ABB RAPID module: Module_OpenholeUD.modx

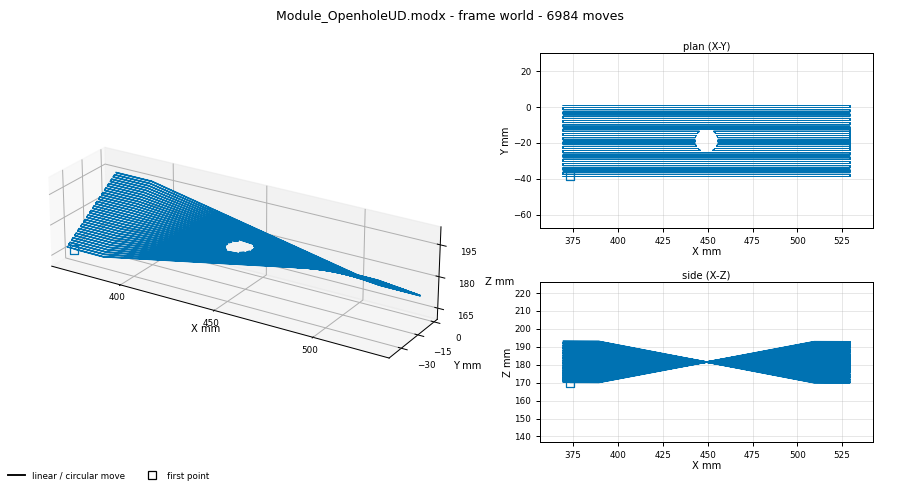
[picture p0: tool path of Module_OpenholeUD.modx in frame world, 6984 of 6984 moves have a stored position in this frame; points joined in program order, loops and branches not executed]
MODULE Module_OpenholeUD

	VAR robtarget OpenholeUD_0 := [[373.31, -38.7, 169.95], [-0.183051, 0.683002, 0.683002, 0.183051], [0,0,0,0], [9E9, 9E9, 9E9, 9E9, 9E9, 9E9]];
	VAR robtarget OpenholeUD_1 := [[377.31, -38.7, 169.94], [-0.183051, 0.683002, 0.683002, 0.183051], [0,0,0,0], [9E9, 9E9, 9E9, 9E9, 9E9, 9E9]];
	VAR robtarget OpenholeUD_2 := [[381.31, -38.7, 169.93], [-0.183051, 0.683002, 0.683002, 0.183051], [0,0,0,0], [9E9, 9E9, 9E9, 9E9, 9E9, 9E9]];
	VAR robtarget OpenholeUD_3 := [[385.31, -38.7, 169.91], [-0.183051, 0.683002, 0.683002, 0.183051], [0,0,0,0], [9E9, 9E9, 9E9, 9E9, 9E9, 9E9]];
	VAR robtarget OpenholeUD_4 := [[389.31, -38.7, 169.9], [-0.126214, 0.695751, 0.665684, 0.238465], [0,0,0,0], [9E9, 9E9, 9E9, 9E9, 9E9, 9E9]];
	VAR robtarget OpenholeUD_5 := [[393.24, -38.7, 170.64], [-0.115233, 0.697654, 0.668744, 0.229742], [0,0,0,0], [9E9, 9E9, 9E9, 9E9, 9E9, 9E9]];
	VAR robtarget OpenholeUD_6 := [[397.17, -38.7, 171.39], [-0.103921, 0.699429, 0.671799, 0.220649], [0,0,0,0], [9E9, 9E9, 9E9, 9E9, 9E9, 9E9]];
	VAR robtarget OpenholeUD_7 := [[401.1, -38.7, 172.13], [-0.092289, 0.701058, 0.674835, 0.211182], [0,0,0,0], [9E9, 9E9, 9E9, 9E9, 9E9, 9E9]];
	VAR robtarget OpenholeUD_8 := [[405.03, -38.7, 172.88], [-0.080349, 0.702527, 0.677838, 0.201336], [0,0,0,0], [9E9, 9E9, 9E9, 9E9, 9E9, 9E9]];
	VAR robtarget OpenholeUD_9 := [[408.96, -38.7, 173.62], [-0.068121, 0.703818, 0.680791, 0.191112], [0,0,0,0], [9E9, 9E9, 9E9, 9E9, 9E9, 9E9]];
	VAR robtarget OpenholeUD_10 := [[412.89, -38.7, 174.36], [-0.055624, 0.704916, 0.683677, 0.180513], [0,0,0,0], [9E9, 9E9, 9E9, 9E9, 9E9, 9E9]];
	VAR robtarget OpenholeUD_11 := [[416.82, -38.7, 175.11], [-0.042884, 0.705805, 0.68648, 0.169546], [0,0,0,0], [9E9, 9E9, 9E9, 9E9, 9E9, 9E9]];
	VAR robtarget OpenholeUD_12 := [[420.75, -38.7, 175.85], [-0.029931, 0.706473, 0.689178, 0.15822], [0,0,0,0], [9E9, 9E9, 9E9, 9E9, 9E9, 9E9]];
	VAR robtarget OpenholeUD_13 := [[424.68, -38.7, 176.59], [-0.016796, 0.706907, 0.691754, 0.14655], [0,0,0,0], [9E9, 9E9, 9E9, 9E9, 9E9, 9E9]];
	VAR robtarget OpenholeUD_14 := [[428.61, -38.7, 177.34], [-0.003517, 0.707098, 0.694187, 0.134555], [0,0,0,0], [9E9, 9E9, 9E9, 9E9, 9E9, 9E9]];
	VAR robtarget OpenholeUD_15 := [[432.54, -38.7, 178.08], [0.009868, 0.707038, 0.696458, 0.122257], [0,0,0,0], [9E9, 9E9, 9E9, 9E9, 9E9, 9E9]];
	VAR robtarget OpenholeUD_16 := [[436.47, -38.7, 178.83], [0.023319, 0.706722, 0.698548, 0.109684], [0,0,0,0], [9E9, 9E9, 9E9, 9E9, 9E9, 9E9]];
	VAR robtarget OpenholeUD_17 := [[440.4, -38.7, 179.57], [0.03679, 0.706149, 0.700441, 0.096866], [0,0,0,0], [9E9, 9E9, 9E9, 9E9, 9E9, 9E9]];
	VAR robtarget OpenholeUD_18 := [[444.33, -38.7, 180.31], [0.05024, 0.70532, 0.702119, 0.083838], [0,0,0,0], [9E9, 9E9, 9E9, 9E9, 9E9, 9E9]];
	VAR robtarget OpenholeUD_19 := [[448.26, -38.7, 181.06], [0.063624, 0.704239, 0.70357, 0.070638], [0,0,0,0], [9E9, 9E9, 9E9, 9E9, 9E9, 9E9]];
	VAR robtarget OpenholeUD_20 := [[452.19, -38.7, 181.8], [0.076899, 0.702913, 0.704781, 0.057307], [0,0,0,0], [9E9, 9E9, 9E9, 9E9, 9E9, 9E9]];
	VAR robtarget OpenholeUD_21 := [[456.12, -38.7, 182.54], [0.090023, 0.701353, 0.705744, 0.043887], [0,0,0,0], [9E9, 9E9, 9E9, 9E9, 9E9, 9E9]];
	VAR robtarget OpenholeUD_22 := [[460.05, -38.7, 183.29], [0.102957, 0.699571, 0.706452, 0.030421], [0,0,0,0], [9E9, 9E9, 9E9, 9E9, 9E9, 9E9]];
	VAR robtarget OpenholeUD_23 := [[463.98, -38.7, 184.03], [0.115664, 0.697583, 0.706903, 0.016955], [0,0,0,0], [9E9, 9E9, 9E9, 9E9, 9E9, 9E9]];
	VAR robtarget OpenholeUD_24 := [[467.91, -38.7, 184.78], [0.128112, 0.695404, 0.707098, 0.003531], [0,0,0,0], [9E9, 9E9, 9E9, 9E9, 9E9, 9E9]];
	VAR robtarget OpenholeUD_25 := [[471.85, -38.7, 185.52], [0.14027, 0.693054, 0.707039, -0.009809], [0,0,0,0], [9E9, 9E9, 9E9, 9E9, 9E9, 9E9]];
	VAR robtarget OpenholeUD_26 := [[475.78, -38.7, 186.26], [0.152115, 0.690551, 0.706732, -0.023024], [0,0,0,0], [9E9, 9E9, 9E9, 9E9, 9E9, 9E9]];
	VAR robtarget OpenholeUD_27 := [[479.71, -38.7, 187.01], [0.163624, 0.687915, 0.706186, -0.036076], [0,0,0,0], [9E9, 9E9, 9E9, 9E9, 9E9, 9E9]];
	VAR robtarget OpenholeUD_28 := [[483.64, -38.7, 187.75], [0.174782, 0.685165, 0.705412, -0.048932], [0,0,0,0], [9E9, 9E9, 9E9, 9E9, 9E9, 9E9]];
	VAR robtarget OpenholeUD_29 := [[487.57, -38.7, 188.49], [0.185577, 0.68232, 0.704422, -0.06156], [0,0,0,0], [9E9, 9E9, 9E9, 9E9, 9E9, 9E9]];
	VAR robtarget OpenholeUD_30 := [[491.5, -38.7, 189.24], [0.195999, 0.6794, 0.703231, -0.073932], [0,0,0,0], [9E9, 9E9, 9E9, 9E9, 9E9, 9E9]];
	VAR robtarget OpenholeUD_31 := [[495.43, -38.7, 189.98], [0.206044, 0.676421, 0.701854, -0.086026], [0,0,0,0], [9E9, 9E9, 9E9, 9E9, 9E9, 9E9]];
	VAR robtarget OpenholeUD_32 := [[499.36, -38.7, 190.73], [0.215711, 0.673401, 0.700308, -0.097822], [0,0,0,0], [9E9, 9E9, 9E9, 9E9, 9E9, 9E9]];
	VAR robtarget OpenholeUD_33 := [[503.29, -38.7, 191.47], [0.225001, 0.670354, 0.698608, -0.109304], [0,0,0,0], [9E9, 9E9, 9E9, 9E9, 9E9, 9E9]];
	VAR robtarget OpenholeUD_34 := [[509.38, -38.7, 192.62], [0.183051, 0.683002, 0.683002, -0.183051], [0,0,0,0], [9E9, 9E9, 9E9, 9E9, 9E9, 9E9]];
	VAR robtarget OpenholeUD_35 := [[513.38, -38.7, 192.61], [0.183051, 0.683002, 0.683002, -0.183051], [0,0,0,0], [9E9, 9E9, 9E9, 9E9, 9E9, 9E9]];
	VAR robtarget OpenholeUD_36 := [[517.38, -38.7, 192.6], [0.183051, 0.683002, 0.683002, -0.183051], [0,0,0,0], [9E9, 9E9, 9E9, 9E9, 9E9, 9E9]];
	VAR robtarget OpenholeUD_37 := [[521.38, -38.7, 192.59], [0.183051, 0.683002, 0.683002, -0.183051], [0,0,0,0], [9E9, 9E9, 9E9, 9E9, 9E9, 9E9]];
	VAR robtarget OpenholeUD_38 := [[529.38, -38.7, 192.56], [0.183051, 0.683002, 0.683002, -0.183051], [0,0,0,0], [9E9, 9E9, 9E9, 9E9, 9E9, 9E9]];
	VAR robtarget OpenholeUD_39 := [[529.38, -38.7, 192.56], [0.183051, 0.683002, 0.683002, -0.183051], [0,0,0,0], [9E9, 9E9, 9E9, 9E9, 9E9, 9E9]];
	VAR robtarget OpenholeUD_40 := [[529.38, -37.5, 191.87], [0.183051, 0.683002, 0.683002, -0.183051], [0,0,0,0], [9E9, 9E9, 9E9, 9E9, 9E9, 9E9]];
	VAR robtarget OpenholeUD_41 := [[525.38, -37.5, 191.88], [0.183051, 0.683002, 0.683002, -0.183051], [0,0,0,0], [9E9, 9E9, 9E9, 9E9, 9E9, 9E9]];
	VAR robtarget OpenholeUD_42 := [[521.38, -37.5, 191.89], [0.183051, 0.683002, 0.683002, -0.183051], [0,0,0,0], [9E9, 9E9, 9E9, 9E9, 9E9, 9E9]];
	VAR robtarget OpenholeUD_43 := [[517.38, -37.5, 191.9], [0.183051, 0.683002, 0.683002, -0.183051], [0,0,0,0], [9E9, 9E9, 9E9, 9E9, 9E9, 9E9]];
	VAR robtarget OpenholeUD_44 := [[509.38, -37.5, 191.93], [0.183051, 0.683002, 0.683002, -0.183051], [0,0,0,0], [9E9, 9E9, 9E9, 9E9, 9E9, 9E9]];
	VAR robtarget OpenholeUD_45 := [[505.44, -37.5, 191.23], [0.226628, 0.669806, 0.697036, -0.118915], [0,0,0,0], [9E9, 9E9, 9E9, 9E9, 9E9, 9E9]];
	VAR robtarget OpenholeUD_46 := [[501.5, -37.5, 190.53], [0.21746, 0.672838, 0.698865, -0.107647], [0,0,0,0], [9E9, 9E9, 9E9, 9E9, 9E9, 9E9]];
	VAR robtarget OpenholeUD_47 := [[497.56, -37.5, 189.83], [0.207916, 0.675848, 0.700552, -0.096055], [0,0,0,0], [9E9, 9E9, 9E9, 9E9, 9E9, 9E9]];
	VAR robtarget OpenholeUD_48 := [[493.63, -37.5, 189.13], [0.197995, 0.678821, 0.702082, -0.084152], [0,0,0,0], [9E9, 9E9, 9E9, 9E9, 9E9, 9E9]];
	VAR robtarget OpenholeUD_49 := [[489.69, -37.5, 188.43], [0.187696, 0.681741, 0.703436, -0.071954], [0,0,0,0], [9E9, 9E9, 9E9, 9E9, 9E9, 9E9]];
	VAR robtarget OpenholeUD_50 := [[485.75, -37.5, 187.73], [0.177023, 0.68459, 0.7046, -0.059484], [0,0,0,0], [9E9, 9E9, 9E9, 9E9, 9E9, 9E9]];
	VAR robtarget OpenholeUD_51 := [[481.81, -37.5, 187.03], [0.165982, 0.68735, 0.705559, -0.046765], [0,0,0,0], [9E9, 9E9, 9E9, 9E9, 9E9, 9E9]];
	VAR robtarget OpenholeUD_52 := [[477.87, -37.5, 186.33], [0.154586, 0.690002, 0.706297, -0.033827], [0,0,0,0], [9E9, 9E9, 9E9, 9E9, 9E9, 9E9]];
	VAR robtarget OpenholeUD_53 := [[473.94, -37.5, 185.63], [0.142847, 0.692528, 0.706804, -0.020702], [0,0,0,0], [9E9, 9E9, 9E9, 9E9, 9E9, 9E9]];
	VAR robtarget OpenholeUD_54 := [[470, -37.5, 184.93], [0.130787, 0.694906, 0.707068, -0.007426], [0,0,0,0], [9E9, 9E9, 9E9, 9E9, 9E9, 9E9]];
	VAR robtarget OpenholeUD_55 := [[466.06, -37.5, 184.23], [0.118427, 0.697119, 0.707082, 0.005963], [0,0,0,0], [9E9, 9E9, 9E9, 9E9, 9E9, 9E9]];
	VAR robtarget OpenholeUD_56 := [[462.12, -37.5, 183.53], [0.105796, 0.699147, 0.70684, 0.019422], [0,0,0,0], [9E9, 9E9, 9E9, 9E9, 9E9, 9E9]];
	VAR robtarget OpenholeUD_57 := [[458.18, -37.5, 182.83], [0.092926, 0.700974, 0.706341, 0.03291], [0,0,0,0], [9E9, 9E9, 9E9, 9E9, 9E9, 9E9]];
	VAR robtarget OpenholeUD_58 := [[454.24, -37.5, 182.13], [0.079851, 0.702584, 0.705584, 0.046383], [0,0,0,0], [9E9, 9E9, 9E9, 9E9, 9E9, 9E9]];
	VAR robtarget OpenholeUD_59 := [[450.31, -37.5, 181.43], [0.06661, 0.703962, 0.704574, 0.059795], [0,0,0,0], [9E9, 9E9, 9E9, 9E9, 9E9, 9E9]];
	VAR robtarget OpenholeUD_60 := [[446.37, -37.5, 180.73], [0.053244, 0.705099, 0.703318, 0.073104], [0,0,0,0], [9E9, 9E9, 9E9, 9E9, 9E9, 9E9]];
	VAR robtarget OpenholeUD_61 := [[442.43, -37.5, 180.03], [0.039796, 0.705986, 0.701825, 0.086268], [0,0,0,0], [9E9, 9E9, 9E9, 9E9, 9E9, 9E9]];
	VAR robtarget OpenholeUD_62 := [[438.49, -37.5, 179.33], [0.02631, 0.706617, 0.700107, 0.099247], [0,0,0,0], [9E9, 9E9, 9E9, 9E9, 9E9, 9E9]];
	VAR robtarget OpenholeUD_63 := [[434.55, -37.5, 178.63], [0.012829, 0.70699, 0.69818, 0.112004], [0,0,0,0], [9E9, 9E9, 9E9, 9E9, 9E9, 9E9]];
	VAR robtarget OpenholeUD_64 := [[430.61, -37.5, 177.93], [-0.000601, 0.707107, 0.696059, 0.124505], [0,0,0,0], [9E9, 9E9, 9E9, 9E9, 9E9, 9E9]];
	VAR robtarget OpenholeUD_65 := [[426.68, -37.5, 177.23], [-0.013941, 0.706969, 0.693763, 0.136721], [0,0,0,0], [9E9, 9E9, 9E9, 9E9, 9E9, 9E9]];
	VAR robtarget OpenholeUD_66 := [[422.74, -37.5, 176.53], [-0.027148, 0.706585, 0.691311, 0.148626], [0,0,0,0], [9E9, 9E9, 9E9, 9E9, 9E9, 9E9]];
	VAR robtarget OpenholeUD_67 := [[418.8, -37.5, 175.83], [-0.040187, 0.705964, 0.688721, 0.160199], [0,0,0,0], [9E9, 9E9, 9E9, 9E9, 9E9, 9E9]];
	VAR robtarget OpenholeUD_68 := [[414.86, -37.5, 175.13], [-0.053022, 0.705116, 0.686013, 0.171422], [0,0,0,0], [9E9, 9E9, 9E9, 9E9, 9E9, 9E9]];
	VAR robtarget OpenholeUD_69 := [[410.92, -37.5, 174.43], [-0.065623, 0.704055, 0.683208, 0.182284], [0,0,0,0], [9E9, 9E9, 9E9, 9E9, 9E9, 9E9]];
	VAR robtarget OpenholeUD_70 := [[406.98, -37.5, 173.73], [-0.077963, 0.702796, 0.680322, 0.192774], [0,0,0,0], [9E9, 9E9, 9E9, 9E9, 9E9, 9E9]];
	VAR robtarget OpenholeUD_71 := [[403.05, -37.5, 173.03], [-0.09002, 0.701353, 0.677374, 0.202889], [0,0,0,0], [9E9, 9E9, 9E9, 9E9, 9E9, 9E9]];
	VAR robtarget OpenholeUD_72 := [[399.11, -37.5, 172.33], [-0.101773, 0.699744, 0.674382, 0.212625], [0,0,0,0], [9E9, 9E9, 9E9, 9E9, 9E9, 9E9]];
	VAR robtarget OpenholeUD_73 := [[395.17, -37.5, 171.63], [-0.113209, 0.697986, 0.671359, 0.221984], [0,0,0,0], [9E9, 9E9, 9E9, 9E9, 9E9, 9E9]];
	VAR robtarget OpenholeUD_74 := [[389.31, -37.5, 170.59], [-0.129603, 0.695128, 0.666839, 0.235215], [0,0,0,0], [9E9, 9E9, 9E9, 9E9, 9E9, 9E9]];
	VAR robtarget OpenholeUD_75 := [[385.31, -37.5, 170.61], [-0.183051, 0.683002, 0.683002, 0.183051], [0,0,0,0], [9E9, 9E9, 9E9, 9E9, 9E9, 9E9]];
	VAR robtarget OpenholeUD_76 := [[381.31, -37.5, 170.62], [-0.183051, 0.683002, 0.683002, 0.183051], [0,0,0,0], [9E9, 9E9, 9E9, 9E9, 9E9, 9E9]];
	VAR robtarget OpenholeUD_77 := [[377.31, -37.5, 170.63], [-0.183051, 0.683002, 0.683002, 0.183051], [0,0,0,0], [9E9, 9E9, 9E9, 9E9, 9E9, 9E9]];
	VAR robtarget OpenholeUD_78 := [[373.31, -37.5, 170.64], [-0.183051, 0.683002, 0.683002, 0.183051], [0,0,0,0], [9E9, 9E9, 9E9, 9E9, 9E9, 9E9]];
	VAR robtarget OpenholeUD_79 := [[369.31, -37.5, 170.66], [-0.183051, 0.683002, 0.683002, 0.183051], [0,0,0,0], [9E9, 9E9, 9E9, 9E9, 9E9, 9E9]];
	VAR robtarget OpenholeUD_80 := [[369.31, -37.5, 170.66], [-0.183051, 0.683002, 0.683002, 0.183051], [0,0,0,0], [9E9, 9E9, 9E9, 9E9, 9E9, 9E9]];
	VAR robtarget OpenholeUD_81 := [[369.31, -36.3, 171.35], [-0.183051, 0.683002, 0.683002, 0.183051], [0,0,0,0], [9E9, 9E9, 9E9, 9E9, 9E9, 9E9]];
	VAR robtarget OpenholeUD_82 := [[373.31, -36.3, 171.34], [-0.183051, 0.683002, 0.683002, 0.183051], [0,0,0,0], [9E9, 9E9, 9E9, 9E9, 9E9, 9E9]];
	VAR robtarget OpenholeUD_83 := [[377.31, -36.3, 171.32], [-0.183051, 0.683002, 0.683002, 0.183051], [0,0,0,0], [9E9, 9E9, 9E9, 9E9, 9E9, 9E9]];
	VAR robtarget OpenholeUD_84 := [[381.31, -36.3, 171.31], [-0.183051, 0.683002, 0.683002, 0.183051], [0,0,0,0], [9E9, 9E9, 9E9, 9E9, 9E9, 9E9]];
	VAR robtarget OpenholeUD_85 := [[385.31, -36.3, 171.3], [-0.183051, 0.683002, 0.683002, 0.183051], [0,0,0,0], [9E9, 9E9, 9E9, 9E9, 9E9, 9E9]];
	VAR robtarget OpenholeUD_86 := [[389.31, -36.3, 171.29], [-0.133, 0.694486, 0.667982, 0.23195], [0,0,0,0], [9E9, 9E9, 9E9, 9E9, 9E9, 9E9]];
	VAR robtarget OpenholeUD_87 := [[393.26, -36.3, 171.94], [-0.122099, 0.696485, 0.671002, 0.22306], [0,0,0,0], [9E9, 9E9, 9E9, 9E9, 9E9, 9E9]];
	VAR robtarget OpenholeUD_88 := [[397.21, -36.3, 172.6], [-0.11086, 0.698362, 0.67401, 0.213799], [0,0,0,0], [9E9, 9E9, 9E9, 9E9, 9E9, 9E9]];
	VAR robtarget OpenholeUD_89 := [[401.15, -36.3, 173.25], [-0.099295, 0.7001, 0.676992, 0.204163], [0,0,0,0], [9E9, 9E9, 9E9, 9E9, 9E9, 9E9]];
	VAR robtarget OpenholeUD_90 := [[405.1, -36.3, 173.91], [-0.087415, 0.701683, 0.679931, 0.194149], [0,0,0,0], [9E9, 9E9, 9E9, 9E9, 9E9, 9E9]];
	VAR robtarget OpenholeUD_91 := [[409.04, -36.3, 174.56], [-0.075237, 0.703093, 0.682813, 0.183758], [0,0,0,0], [9E9, 9E9, 9E9, 9E9, 9E9, 9E9]];
	VAR robtarget OpenholeUD_92 := [[412.99, -36.3, 175.22], [-0.062782, 0.704314, 0.685619, 0.172994], [0,0,0,0], [9E9, 9E9, 9E9, 9E9, 9E9, 9E9]];
	VAR robtarget OpenholeUD_93 := [[416.94, -36.3, 175.88], [-0.050075, 0.705331, 0.688331, 0.161866], [0,0,0,0], [9E9, 9E9, 9E9, 9E9, 9E9, 9E9]];
	VAR robtarget OpenholeUD_94 := [[420.88, -36.3, 176.53], [-0.037144, 0.706131, 0.69093, 0.150384], [0,0,0,0], [9E9, 9E9, 9E9, 9E9, 9E9, 9E9]];
	VAR robtarget OpenholeUD_95 := [[424.83, -36.3, 177.19], [-0.024021, 0.706699, 0.693397, 0.138564], [0,0,0,0], [9E9, 9E9, 9E9, 9E9, 9E9, 9E9]];
	VAR robtarget OpenholeUD_96 := [[428.77, -36.3, 177.84], [-0.010743, 0.707025, 0.695713, 0.126426], [0,0,0,0], [9E9, 9E9, 9E9, 9E9, 9E9, 9E9]];
	VAR robtarget OpenholeUD_97 := [[432.72, -36.3, 178.5], [0.002652, 0.707102, 0.697858, 0.113995], [0,0,0,0], [9E9, 9E9, 9E9, 9E9, 9E9, 9E9]];
	VAR robtarget OpenholeUD_98 := [[436.67, -36.3, 179.15], [0.016123, 0.706923, 0.699813, 0.101298], [0,0,0,0], [9E9, 9E9, 9E9, 9E9, 9E9, 9E9]];
	VAR robtarget OpenholeUD_99 := [[440.61, -36.3, 179.81], [0.029627, 0.706486, 0.701563, 0.088368], [0,0,0,0], [9E9, 9E9, 9E9, 9E9, 9E9, 9E9]];
	VAR robtarget OpenholeUD_100 := [[444.56, -36.3, 180.47], [0.04312, 0.705791, 0.703092, 0.075241], [0,0,0,0], [9E9, 9E9, 9E9, 9E9, 9E9, 9E9]];
	VAR robtarget OpenholeUD_101 := [[448.5, -36.3, 181.12], [0.056557, 0.704841, 0.704387, 0.061957], [0,0,0,0], [9E9, 9E9, 9E9, 9E9, 9E9, 9E9]];
	VAR robtarget OpenholeUD_102 := [[452.45, -36.3, 181.78], [0.069895, 0.703644, 0.705438, 0.048555], [0,0,0,0], [9E9, 9E9, 9E9, 9E9, 9E9, 9E9]];
	VAR robtarget OpenholeUD_103 := [[456.39, -36.3, 182.43], [0.083091, 0.702208, 0.706236, 0.03508], [0,0,0,0], [9E9, 9E9, 9E9, 9E9, 9E9, 9E9]];
	VAR robtarget OpenholeUD_104 := [[460.34, -36.3, 183.09], [0.096106, 0.700545, 0.706778, 0.021577], [0,0,0,0], [9E9, 9E9, 9E9, 9E9, 9E9, 9E9]];
	VAR robtarget OpenholeUD_105 := [[464.29, -36.3, 183.74], [0.108902, 0.69867, 0.707061, 0.008088], [0,0,0,0], [9E9, 9E9, 9E9, 9E9, 9E9, 9E9]];
	VAR robtarget OpenholeUD_106 := [[468.23, -36.3, 184.4], [0.121445, 0.6966, 0.707087, -0.005342], [0,0,0,0], [9E9, 9E9, 9E9, 9E9, 9E9, 9E9]];
	VAR robtarget OpenholeUD_107 := [[472.18, -36.3, 185.06], [0.133705, 0.694351, 0.70686, -0.018672], [0,0,0,0], [9E9, 9E9, 9E9, 9E9, 9E9, 9E9]];
	VAR robtarget OpenholeUD_108 := [[476.12, -36.3, 185.71], [0.145657, 0.691942, 0.706389, -0.031861], [0,0,0,0], [9E9, 9E9, 9E9, 9E9, 9E9, 9E9]];
	VAR robtarget OpenholeUD_109 := [[480.07, -36.3, 186.37], [0.157278, 0.689394, 0.705682, -0.044873], [0,0,0,0], [9E9, 9E9, 9E9, 9E9, 9E9, 9E9]];
	VAR robtarget OpenholeUD_110 := [[484.02, -36.3, 187.02], [0.168551, 0.686724, 0.704751, -0.057673], [0,0,0,0], [9E9, 9E9, 9E9, 9E9, 9E9, 9E9]];
	VAR robtarget OpenholeUD_111 := [[487.96, -36.3, 187.68], [0.179463, 0.683954, 0.70361, -0.070232], [0,0,0,0], [9E9, 9E9, 9E9, 9E9, 9E9, 9E9]];
	VAR robtarget OpenholeUD_112 := [[491.91, -36.3, 188.33], [0.190006, 0.6811, 0.702275, -0.082524], [0,0,0,0], [9E9, 9E9, 9E9, 9E9, 9E9, 9E9]];
	VAR robtarget OpenholeUD_113 := [[495.85, -36.3, 188.99], [0.200172, 0.678182, 0.70076, -0.094526], [0,0,0,0], [9E9, 9E9, 9E9, 9E9, 9E9, 9E9]];
	VAR robtarget OpenholeUD_114 := [[499.8, -36.3, 189.65], [0.209961, 0.675216, 0.699083, -0.10622], [0,0,0,0], [9E9, 9E9, 9E9, 9E9, 9E9, 9E9]];
	VAR robtarget OpenholeUD_115 := [[503.75, -36.3, 190.3], [0.219374, 0.672217, 0.69726, -0.117592], [0,0,0,0], [9E9, 9E9, 9E9, 9E9, 9E9, 9E9]];
	VAR robtarget OpenholeUD_116 := [[509.38, -36.3, 191.24], [0.183051, 0.683002, 0.683002, -0.183051], [0,0,0,0], [9E9, 9E9, 9E9, 9E9, 9E9, 9E9]];
	VAR robtarget OpenholeUD_117 := [[513.38, -36.3, 191.22], [0.183051, 0.683002, 0.683002, -0.183051], [0,0,0,0], [9E9, 9E9, 9E9, 9E9, 9E9, 9E9]];
	VAR robtarget OpenholeUD_118 := [[517.38, -36.3, 191.21], [0.183051, 0.683002, 0.683002, -0.183051], [0,0,0,0], [9E9, 9E9, 9E9, 9E9, 9E9, 9E9]];
	VAR robtarget OpenholeUD_119 := [[521.38, -36.3, 191.2], [0.183051, 0.683002, 0.683002, -0.183051], [0,0,0,0], [9E9, 9E9, 9E9, 9E9, 9E9, 9E9]];
	VAR robtarget OpenholeUD_120 := [[525.38, -36.3, 191.19], [0.183051, 0.683002, 0.683002, -0.183051], [0,0,0,0], [9E9, 9E9, 9E9, 9E9, 9E9, 9E9]];
	VAR robtarget OpenholeUD_121 := [[529.38, -36.3, 191.17], [0.183051, 0.683002, 0.683002, -0.183051], [0,0,0,0], [9E9, 9E9, 9E9, 9E9, 9E9, 9E9]];
	VAR robtarget OpenholeUD_122 := [[529.38, -36.3, 191.17], [0.183051, 0.683002, 0.683002, -0.183051], [0,0,0,0], [9E9, 9E9, 9E9, 9E9, 9E9, 9E9]];
	VAR robtarget OpenholeUD_123 := [[529.38, -35.1, 190.48], [0.183051, 0.683002, 0.683002, -0.183051], [0,0,0,0], [9E9, 9E9, 9E9, 9E9, 9E9, 9E9]];
	VAR robtarget OpenholeUD_124 := [[525.38, -35.1, 190.49], [0.183051, 0.683002, 0.683002, -0.183051], [0,0,0,0], [9E9, 9E9, 9E9, 9E9, 9E9, 9E9]];
	VAR robtarget OpenholeUD_125 := [[521.38, -35.1, 190.51], [0.183051, 0.683002, 0.683002, -0.183051], [0,0,0,0], [9E9, 9E9, 9E9, 9E9, 9E9, 9E9]];
	VAR robtarget OpenholeUD_126 := [[517.38, -35.1, 190.52], [0.183051, 0.683002, 0.683002, -0.183051], [0,0,0,0], [9E9, 9E9, 9E9, 9E9, 9E9, 9E9]];
	VAR robtarget OpenholeUD_127 := [[513.38, -35.1, 190.53], [0.183051, 0.683002, 0.683002, -0.183051], [0,0,0,0], [9E9, 9E9, 9E9, 9E9, 9E9, 9E9]];
	VAR robtarget OpenholeUD_128 := [[509.38, -35.1, 190.54], [0.183051, 0.683002, 0.683002, -0.183051], [0,0,0,0], [9E9, 9E9, 9E9, 9E9, 9E9, 9E9]];
	VAR robtarget OpenholeUD_129 := [[505.42, -35.1, 189.93], [0.219922, 0.672037, 0.695827, -0.125794], [0,0,0,0], [9E9, 9E9, 9E9, 9E9, 9E9, 9E9]];
	VAR robtarget OpenholeUD_130 := [[501.47, -35.1, 189.32], [0.210587, 0.675021, 0.697758, -0.114605], [0,0,0,0], [9E9, 9E9, 9E9, 9E9, 9E9, 9E9]];
	VAR robtarget OpenholeUD_131 := [[497.52, -35.1, 188.71], [0.200875, 0.677974, 0.699552, -0.103084], [0,0,0,0], [9E9, 9E9, 9E9, 9E9, 9E9, 9E9]];
	VAR robtarget OpenholeUD_132 := [[493.56, -35.1, 188.1], [0.190787, 0.680882, 0.701195, -0.091245], [0,0,0,0], [9E9, 9E9, 9E9, 9E9, 9E9, 9E9]];
	VAR robtarget OpenholeUD_133 := [[489.61, -35.1, 187.49], [0.180322, 0.683728, 0.702668, -0.079104], [0,0,0,0], [9E9, 9E9, 9E9, 9E9, 9E9, 9E9]];
	VAR robtarget OpenholeUD_134 := [[485.66, -35.1, 186.88], [0.169486, 0.686494, 0.703956, -0.066681], [0,0,0,0], [9E9, 9E9, 9E9, 9E9, 9E9, 9E9]];
	VAR robtarget OpenholeUD_135 := [[481.7, -35.1, 186.27], [0.158287, 0.689163, 0.705042, -0.054001], [0,0,0,0], [9E9, 9E9, 9E9, 9E9, 9E9, 9E9]];
	VAR robtarget OpenholeUD_136 := [[477.75, -35.1, 185.65], [0.146736, 0.691714, 0.705912, -0.041091], [0,0,0,0], [9E9, 9E9, 9E9, 9E9, 9E9, 9E9]];
	VAR robtarget OpenholeUD_137 := [[473.8, -35.1, 185.04], [0.134851, 0.694129, 0.706553, -0.027983], [0,0,0,0], [9E9, 9E9, 9E9, 9E9, 9E9, 9E9]];
	VAR robtarget OpenholeUD_138 := [[469.85, -35.1, 184.43], [0.122651, 0.696388, 0.706954, -0.014713], [0,0,0,0], [9E9, 9E9, 9E9, 9E9, 9E9, 9E9]];
	VAR robtarget OpenholeUD_139 := [[465.89, -35.1, 183.82], [0.110161, 0.698473, 0.707106, -0.001319], [0,0,0,0], [9E9, 9E9, 9E9, 9E9, 9E9, 9E9]];
	VAR robtarget OpenholeUD_140 := [[461.94, -35.1, 183.21], [0.097411, 0.700365, 0.707002, 0.012157], [0,0,0,0], [9E9, 9E9, 9E9, 9E9, 9E9, 9E9]];
	VAR robtarget OpenholeUD_141 := [[457.99, -35.1, 182.6], [0.084432, 0.702048, 0.706641, 0.025672], [0,0,0,0], [9E9, 9E9, 9E9, 9E9, 9E9, 9E9]];
	VAR robtarget OpenholeUD_142 := [[454.03, -35.1, 181.99], [0.071263, 0.703507, 0.70602, 0.039183], [0,0,0,0], [9E9, 9E9, 9E9, 9E9, 9E9, 9E9]];
	VAR robtarget OpenholeUD_143 := [[450.08, -35.1, 181.37], [0.057941, 0.704729, 0.705144, 0.052646], [0,0,0,0], [9E9, 9E9, 9E9, 9E9, 9E9, 9E9]];
	VAR robtarget OpenholeUD_144 := [[446.13, -35.1, 180.76], [0.04451, 0.705705, 0.704019, 0.066015], [0,0,0,0], [9E9, 9E9, 9E9, 9E9, 9E9, 9E9]];
	VAR robtarget OpenholeUD_145 := [[442.17, -35.1, 180.15], [0.031011, 0.706426, 0.702652, 0.079248], [0,0,0,0], [9E9, 9E9, 9E9, 9E9, 9E9, 9E9]];
	VAR robtarget OpenholeUD_146 := [[438.22, -35.1, 179.54], [0.017491, 0.70689, 0.701056, 0.092306], [0,0,0,0], [9E9, 9E9, 9E9, 9E9, 9E9, 9E9]];
	VAR robtarget OpenholeUD_147 := [[434.27, -35.1, 178.93], [0.003993, 0.707096, 0.699245, 0.105149], [0,0,0,0], [9E9, 9E9, 9E9, 9E9, 9E9, 9E9]];
	VAR robtarget OpenholeUD_148 := [[430.32, -35.1, 178.32], [-0.009439, 0.707044, 0.697235, 0.117745], [0,0,0,0], [9E9, 9E9, 9E9, 9E9, 9E9, 9E9]];
	VAR robtarget OpenholeUD_149 := [[426.36, -35.1, 177.71], [-0.022763, 0.70674, 0.695042, 0.130062], [0,0,0,0], [9E9, 9E9, 9E9, 9E9, 9E9, 9E9]];
	VAR robtarget OpenholeUD_150 := [[422.41, -35.1, 177.1], [-0.035941, 0.706193, 0.692687, 0.142074], [0,0,0,0], [9E9, 9E9, 9E9, 9E9, 9E9, 9E9]];
	VAR robtarget OpenholeUD_151 := [[418.46, -35.1, 176.48], [-0.048934, 0.705412, 0.690187, 0.153758], [0,0,0,0], [9E9, 9E9, 9E9, 9E9, 9E9, 9E9]];
	VAR robtarget OpenholeUD_152 := [[414.5, -35.1, 175.87], [-0.061709, 0.704409, 0.687563, 0.165097], [0,0,0,0], [9E9, 9E9, 9E9, 9E9, 9E9, 9E9]];
	VAR robtarget OpenholeUD_153 := [[410.55, -35.1, 175.26], [-0.074238, 0.703199, 0.684833, 0.176077], [0,0,0,0], [9E9, 9E9, 9E9, 9E9, 9E9, 9E9]];
	VAR robtarget OpenholeUD_154 := [[406.6, -35.1, 174.65], [-0.086493, 0.701797, 0.682017, 0.186689], [0,0,0,0], [9E9, 9E9, 9E9, 9E9, 9E9, 9E9]];
	VAR robtarget OpenholeUD_155 := [[402.64, -35.1, 174.04], [-0.098454, 0.700219, 0.679132, 0.196926], [0,0,0,0], [9E9, 9E9, 9E9, 9E9, 9E9, 9E9]];
	VAR robtarget OpenholeUD_156 := [[398.69, -35.1, 173.43], [-0.110103, 0.698482, 0.676195, 0.206786], [0,0,0,0], [9E9, 9E9, 9E9, 9E9, 9E9, 9E9]];
	VAR robtarget OpenholeUD_157 := [[394.74, -35.1, 172.82], [-0.121425, 0.696603, 0.673222, 0.216269], [0,0,0,0], [9E9, 9E9, 9E9, 9E9, 9E9, 9E9]];
	VAR robtarget OpenholeUD_158 := [[389.32, -35.1, 171.98], [-0.136403, 0.693826, 0.669112, 0.228669], [0,0,0,0], [9E9, 9E9, 9E9, 9E9, 9E9, 9E9]];
	VAR robtarget OpenholeUD_159 := [[385.32, -35.1, 171.99], [-0.183051, 0.683002, 0.683002, 0.183051], [0,0,0,0], [9E9, 9E9, 9E9, 9E9, 9E9, 9E9]];
	VAR robtarget OpenholeUD_160 := [[381.32, -35.1, 172], [-0.183051, 0.683002, 0.683002, 0.183051], [0,0,0,0], [9E9, 9E9, 9E9, 9E9, 9E9, 9E9]];
	VAR robtarget OpenholeUD_161 := [[377.32, -35.1, 172.02], [-0.183051, 0.683002, 0.683002, 0.183051], [0,0,0,0], [9E9, 9E9, 9E9, 9E9, 9E9, 9E9]];
	VAR robtarget OpenholeUD_162 := [[373.32, -35.1, 172.03], [-0.183051, 0.683002, 0.683002, 0.183051], [0,0,0,0], [9E9, 9E9, 9E9, 9E9, 9E9, 9E9]];
	VAR robtarget OpenholeUD_163 := [[369.32, -35.1, 172.04], [-0.183051, 0.683002, 0.683002, 0.183051], [0,0,0,0], [9E9, 9E9, 9E9, 9E9, 9E9, 9E9]];
	VAR robtarget OpenholeUD_164 := [[369.32, -35.1, 172.04], [-0.183051, 0.683002, 0.683002, 0.183051], [0,0,0,0], [9E9, 9E9, 9E9, 9E9, 9E9, 9E9]];
	VAR robtarget OpenholeUD_165 := [[369.32, -33.9, 172.73], [-0.183051, 0.683002, 0.683002, 0.183051], [0,0,0,0], [9E9, 9E9, 9E9, 9E9, 9E9, 9E9]];
	VAR robtarget OpenholeUD_166 := [[373.32, -33.9, 172.72], [-0.183051, 0.683002, 0.683002, 0.183051], [0,0,0,0], [9E9, 9E9, 9E9, 9E9, 9E9, 9E9]];
	VAR robtarget OpenholeUD_167 := [[377.32, -33.9, 172.71], [-0.183051, 0.683002, 0.683002, 0.183051], [0,0,0,0], [9E9, 9E9, 9E9, 9E9, 9E9, 9E9]];
	VAR robtarget OpenholeUD_168 := [[381.32, -33.9, 172.7], [-0.183051, 0.683002, 0.683002, 0.183051], [0,0,0,0], [9E9, 9E9, 9E9, 9E9, 9E9, 9E9]];
	VAR robtarget OpenholeUD_169 := [[385.32, -33.9, 172.68], [-0.183051, 0.683002, 0.683002, 0.183051], [0,0,0,0], [9E9, 9E9, 9E9, 9E9, 9E9, 9E9]];
	VAR robtarget OpenholeUD_170 := [[389.32, -33.9, 172.67], [-0.139812, 0.693147, 0.670229, 0.225375], [0,0,0,0], [9E9, 9E9, 9E9, 9E9, 9E9, 9E9]];
	VAR robtarget OpenholeUD_171 := [[393.28, -33.9, 173.24], [-0.128999, 0.69524, 0.673206, 0.216319], [0,0,0,0], [9E9, 9E9, 9E9, 9E9, 9E9, 9E9]];
	VAR robtarget OpenholeUD_172 := [[397.24, -33.9, 173.81], [-0.117844, 0.697218, 0.676162, 0.206892], [0,0,0,0], [9E9, 9E9, 9E9, 9E9, 9E9, 9E9]];
	VAR robtarget OpenholeUD_173 := [[401.2, -33.9, 174.37], [-0.106355, 0.699063, 0.679084, 0.19709], [0,0,0,0], [9E9, 9E9, 9E9, 9E9, 9E9, 9E9]];
	VAR robtarget OpenholeUD_174 := [[405.16, -33.9, 174.94], [-0.094544, 0.700758, 0.681956, 0.18691], [0,0,0,0], [9E9, 9E9, 9E9, 9E9, 9E9, 9E9]];
	VAR robtarget OpenholeUD_175 := [[409.12, -33.9, 175.5], [-0.082427, 0.702286, 0.684762, 0.176356], [0,0,0,0], [9E9, 9E9, 9E9, 9E9, 9E9, 9E9]];
	VAR robtarget OpenholeUD_176 := [[413.08, -33.9, 176.07], [-0.070025, 0.703631, 0.687482, 0.165432], [0,0,0,0], [9E9, 9E9, 9E9, 9E9, 9E9, 9E9]];
	VAR robtarget OpenholeUD_177 := [[417.04, -33.9, 176.64], [-0.05736, 0.704776, 0.6901, 0.154148], [0,0,0,0], [9E9, 9E9, 9E9, 9E9, 9E9, 9E9]];
	VAR robtarget OpenholeUD_178 := [[421, -33.9, 177.2], [-0.044462, 0.705708, 0.692596, 0.142515], [0,0,0,0], [9E9, 9E9, 9E9, 9E9, 9E9, 9E9]];
	VAR robtarget OpenholeUD_179 := [[424.96, -33.9, 177.77], [-0.031361, 0.706411, 0.694951, 0.130552], [0,0,0,0], [9E9, 9E9, 9E9, 9E9, 9E9, 9E9]];
	VAR robtarget OpenholeUD_180 := [[428.92, -33.9, 178.34], [-0.018093, 0.706875, 0.697144, 0.118278], [0,0,0,0], [9E9, 9E9, 9E9, 9E9, 9E9, 9E9]];
	VAR robtarget OpenholeUD_181 := [[432.88, -33.9, 178.9], [-0.004697, 0.707091, 0.699159, 0.105721], [0,0,0,0], [9E9, 9E9, 9E9, 9E9, 9E9, 9E9]];
	VAR robtarget OpenholeUD_182 := [[436.83, -33.9, 179.47], [0.008787, 0.707052, 0.700976, 0.092909], [0,0,0,0], [9E9, 9E9, 9E9, 9E9, 9E9, 9E9]];
	VAR robtarget OpenholeUD_183 := [[440.79, -33.9, 180.04], [0.022315, 0.706755, 0.702581, 0.079877], [0,0,0,0], [9E9, 9E9, 9E9, 9E9, 9E9, 9E9]];
	VAR robtarget OpenholeUD_184 := [[444.75, -33.9, 180.6], [0.035844, 0.706198, 0.703958, 0.06666], [0,0,0,0], [9E9, 9E9, 9E9, 9E9, 9E9, 9E9]];
	VAR robtarget OpenholeUD_185 := [[448.71, -33.9, 181.17], [0.049328, 0.705384, 0.705095, 0.053301], [0,0,0,0], [9E9, 9E9, 9E9, 9E9, 9E9, 9E9]];
	VAR robtarget OpenholeUD_186 := [[452.67, -33.9, 181.74], [0.062723, 0.704319, 0.705984, 0.039839], [0,0,0,0], [9E9, 9E9, 9E9, 9E9, 9E9, 9E9]];
	VAR robtarget OpenholeUD_187 := [[456.63, -33.9, 182.3], [0.075987, 0.703012, 0.706617, 0.026321], [0,0,0,0], [9E9, 9E9, 9E9, 9E9, 9E9, 9E9]];
	VAR robtarget OpenholeUD_188 := [[460.59, -33.9, 182.87], [0.089079, 0.701473, 0.706991, 0.012789], [0,0,0,0], [9E9, 9E9, 9E9, 9E9, 9E9, 9E9]];
	VAR robtarget OpenholeUD_189 := [[464.55, -33.9, 183.44], [0.101961, 0.699717, 0.707106, -0.000711], [0,0,0,0], [9E9, 9E9, 9E9, 9E9, 9E9, 9E9]];
	VAR robtarget OpenholeUD_190 := [[468.51, -33.9, 184], [0.114598, 0.697759, 0.706965, -0.014137], [0,0,0,0], [9E9, 9E9, 9E9, 9E9, 9E9, 9E9]];
	VAR robtarget OpenholeUD_191 := [[472.47, -33.9, 184.57], [0.126959, 0.695616, 0.706574, -0.027446], [0,0,0,0], [9E9, 9E9, 9E9, 9E9, 9E9, 9E9]];
	VAR robtarget OpenholeUD_192 := [[476.43, -33.9, 185.14], [0.139018, 0.693307, 0.70594, -0.040599], [0,0,0,0], [9E9, 9E9, 9E9, 9E9, 9E9, 9E9]];
	VAR robtarget OpenholeUD_193 := [[480.39, -33.9, 185.7], [0.150751, 0.69085, 0.705075, -0.05356], [0,0,0,0], [9E9, 9E9, 9E9, 9E9, 9E9, 9E9]];
	VAR robtarget OpenholeUD_194 := [[484.35, -33.9, 186.27], [0.16214, 0.688266, 0.703992, -0.066296], [0,0,0,0], [9E9, 9E9, 9E9, 9E9, 9E9, 9E9]];
	VAR robtarget OpenholeUD_195 := [[488.31, -33.9, 186.84], [0.173173, 0.685574, 0.702705, -0.078778], [0,0,0,0], [9E9, 9E9, 9E9, 9E9, 9E9, 9E9]];
	VAR robtarget OpenholeUD_196 := [[492.27, -33.9, 187.4], [0.183837, 0.682791, 0.701229, -0.090981], [0,0,0,0], [9E9, 9E9, 9E9, 9E9, 9E9, 9E9]];
	VAR robtarget OpenholeUD_197 := [[496.23, -33.9, 187.97], [0.194128, 0.679937, 0.699582, -0.102883], [0,0,0,0], [9E9, 9E9, 9E9, 9E9, 9E9, 9E9]];
	VAR robtarget OpenholeUD_198 := [[500.19, -33.9, 188.54], [0.204043, 0.677028, 0.69778, -0.114469], [0,0,0,0], [9E9, 9E9, 9E9, 9E9, 9E9, 9E9]];
	VAR robtarget OpenholeUD_199 := [[504.15, -33.9, 189.1], [0.213581, 0.67408, 0.69584, -0.125723], [0,0,0,0], [9E9, 9E9, 9E9, 9E9, 9E9, 9E9]];
	VAR robtarget OpenholeUD_200 := [[509.37, -33.9, 189.85], [0.183051, 0.683002, 0.683002, -0.183051], [0,0,0,0], [9E9, 9E9, 9E9, 9E9, 9E9, 9E9]];
	VAR robtarget OpenholeUD_201 := [[513.37, -33.9, 189.84], [0.183051, 0.683002, 0.683002, -0.183051], [0,0,0,0], [9E9, 9E9, 9E9, 9E9, 9E9, 9E9]];
	VAR robtarget OpenholeUD_202 := [[517.37, -33.9, 189.83], [0.183051, 0.683002, 0.683002, -0.183051], [0,0,0,0], [9E9, 9E9, 9E9, 9E9, 9E9, 9E9]];
	VAR robtarget OpenholeUD_203 := [[521.37, -33.9, 189.81], [0.183051, 0.683002, 0.683002, -0.183051], [0,0,0,0], [9E9, 9E9, 9E9, 9E9, 9E9, 9E9]];
	VAR robtarget OpenholeUD_204 := [[525.37, -33.9, 189.8], [0.183051, 0.683002, 0.683002, -0.183051], [0,0,0,0], [9E9, 9E9, 9E9, 9E9, 9E9, 9E9]];
	VAR robtarget OpenholeUD_205 := [[529.37, -33.9, 189.79], [0.183051, 0.683002, 0.683002, -0.183051], [0,0,0,0], [9E9, 9E9, 9E9, 9E9, 9E9, 9E9]];
	VAR robtarget OpenholeUD_206 := [[529.37, -33.9, 189.79], [0.183051, 0.683002, 0.683002, -0.183051], [0,0,0,0], [9E9, 9E9, 9E9, 9E9, 9E9, 9E9]];
	VAR robtarget OpenholeUD_207 := [[529.37, -32.7, 189.1], [0.183051, 0.683002, 0.683002, -0.183051], [0,0,0,0], [9E9, 9E9, 9E9, 9E9, 9E9, 9E9]];
	VAR robtarget OpenholeUD_208 := [[525.37, -32.7, 189.11], [0.183051, 0.683002, 0.683002, -0.183051], [0,0,0,0], [9E9, 9E9, 9E9, 9E9, 9E9, 9E9]];
	VAR robtarget OpenholeUD_209 := [[521.37, -32.7, 189.12], [0.183051, 0.683002, 0.683002, -0.183051], [0,0,0,0], [9E9, 9E9, 9E9, 9E9, 9E9, 9E9]];
	VAR robtarget OpenholeUD_210 := [[517.37, -32.7, 189.13], [0.183051, 0.683002, 0.683002, -0.183051], [0,0,0,0], [9E9, 9E9, 9E9, 9E9, 9E9, 9E9]];
	VAR robtarget OpenholeUD_211 := [[513.37, -32.7, 189.15], [0.183051, 0.683002, 0.683002, -0.183051], [0,0,0,0], [9E9, 9E9, 9E9, 9E9, 9E9, 9E9]];
	VAR robtarget OpenholeUD_212 := [[509.37, -32.7, 189.16], [0.183051, 0.683002, 0.683002, -0.183051], [0,0,0,0], [9E9, 9E9, 9E9, 9E9, 9E9, 9E9]];
	VAR robtarget OpenholeUD_213 := [[505.41, -32.7, 188.64], [0.213161, 0.674213, 0.694543, -0.132705], [0,0,0,0], [9E9, 9E9, 9E9, 9E9, 9E9, 9E9]];
	VAR robtarget OpenholeUD_214 := [[501.44, -32.7, 188.11], [0.20366, 0.677143, 0.696572, -0.121603], [0,0,0,0], [9E9, 9E9, 9E9, 9E9, 9E9, 9E9]];
	VAR robtarget OpenholeUD_215 := [[497.47, -32.7, 187.59], [0.193784, 0.680035, 0.698473, -0.110164], [0,0,0,0], [9E9, 9E9, 9E9, 9E9, 9E9, 9E9]];
	VAR robtarget OpenholeUD_216 := [[493.51, -32.7, 187.07], [0.183532, 0.682873, 0.700227, -0.098399], [0,0,0,0], [9E9, 9E9, 9E9, 9E9, 9E9, 9E9]];
	VAR robtarget OpenholeUD_217 := [[489.54, -32.7, 186.55], [0.172905, 0.685641, 0.701818, -0.086325], [0,0,0,0], [9E9, 9E9, 9E9, 9E9, 9E9, 9E9]];
	VAR robtarget OpenholeUD_218 := [[485.58, -32.7, 186.03], [0.161911, 0.68832, 0.703228, -0.073959], [0,0,0,0], [9E9, 9E9, 9E9, 9E9, 9E9, 9E9]];
	VAR robtarget OpenholeUD_219 := [[481.61, -32.7, 185.51], [0.150558, 0.690892, 0.704442, -0.061327], [0,0,0,0], [9E9, 9E9, 9E9, 9E9, 9E9, 9E9]];
	VAR robtarget OpenholeUD_220 := [[477.64, -32.7, 184.98], [0.13886, 0.693338, 0.705445, -0.048454], [0,0,0,0], [9E9, 9E9, 9E9, 9E9, 9E9, 9E9]];
	VAR robtarget OpenholeUD_221 := [[473.68, -32.7, 184.46], [0.126833, 0.695639, 0.706221, -0.035374], [0,0,0,0], [9E9, 9E9, 9E9, 9E9, 9E9, 9E9]];
	VAR robtarget OpenholeUD_222 := [[469.71, -32.7, 183.94], [0.114501, 0.697775, 0.706761, -0.02212], [0,0,0,0], [9E9, 9E9, 9E9, 9E9, 9E9, 9E9]];
	VAR robtarget OpenholeUD_223 := [[465.75, -32.7, 183.42], [0.101889, 0.699728, 0.707053, -0.00873], [0,0,0,0], [9E9, 9E9, 9E9, 9E9, 9E9, 9E9]];
	VAR robtarget OpenholeUD_224 := [[461.78, -32.7, 182.9], [0.089027, 0.70148, 0.707091, 0.004754], [0,0,0,0], [9E9, 9E9, 9E9, 9E9, 9E9, 9E9]];
	VAR robtarget OpenholeUD_225 := [[457.82, -32.7, 182.38], [0.07595, 0.703016, 0.70687, 0.018289], [0,0,0,0], [9E9, 9E9, 9E9, 9E9, 9E9, 9E9]];
	VAR robtarget OpenholeUD_226 := [[453.85, -32.7, 181.85], [0.062695, 0.704322, 0.70639, 0.031831], [0,0,0,0], [9E9, 9E9, 9E9, 9E9, 9E9, 9E9]];
	VAR robtarget OpenholeUD_227 := [[449.88, -32.7, 181.33], [0.049303, 0.705386, 0.705652, 0.045336], [0,0,0,0], [9E9, 9E9, 9E9, 9E9, 9E9, 9E9]];
	VAR robtarget OpenholeUD_228 := [[445.92, -32.7, 180.81], [0.035816, 0.706199, 0.704661, 0.05876], [0,0,0,0], [9E9, 9E9, 9E9, 9E9, 9E9, 9E9]];
	VAR robtarget OpenholeUD_229 := [[441.95, -32.7, 180.29], [0.022279, 0.706756, 0.703426, 0.072058], [0,0,0,0], [9E9, 9E9, 9E9, 9E9, 9E9, 9E9]];
	VAR robtarget OpenholeUD_230 := [[437.99, -32.7, 179.77], [0.008736, 0.707053, 0.701956, 0.08519], [0,0,0,0], [9E9, 9E9, 9E9, 9E9, 9E9, 9E9]];
	VAR robtarget OpenholeUD_231 := [[434.02, -32.7, 179.25], [-0.004769, 0.707091, 0.700266, 0.098118], [0,0,0,0], [9E9, 9E9, 9E9, 9E9, 9E9, 9E9]];
	VAR robtarget OpenholeUD_232 := [[430.05, -32.7, 178.72], [-0.018192, 0.706873, 0.698371, 0.110806], [0,0,0,0], [9E9, 9E9, 9E9, 9E9, 9E9, 9E9]];
	VAR robtarget OpenholeUD_233 := [[426.09, -32.7, 178.2], [-0.031491, 0.706405, 0.696287, 0.123222], [0,0,0,0], [9E9, 9E9, 9E9, 9E9, 9E9, 9E9]];
	VAR robtarget OpenholeUD_234 := [[422.12, -32.7, 177.68], [-0.044628, 0.705697, 0.694034, 0.13534], [0,0,0,0], [9E9, 9E9, 9E9, 9E9, 9E9, 9E9]];
	VAR robtarget OpenholeUD_235 := [[418.16, -32.7, 177.16], [-0.057566, 0.70476, 0.691629, 0.147137], [0,0,0,0], [9E9, 9E9, 9E9, 9E9, 9E9, 9E9]];
	VAR robtarget OpenholeUD_236 := [[414.19, -32.7, 176.64], [-0.070274, 0.703606, 0.689092, 0.158592], [0,0,0,0], [9E9, 9E9, 9E9, 9E9, 9E9, 9E9]];
	VAR robtarget OpenholeUD_237 := [[410.23, -32.7, 176.12], [-0.082721, 0.702252, 0.686443, 0.169693], [0,0,0,0], [9E9, 9E9, 9E9, 9E9, 9E9, 9E9]];
	VAR robtarget OpenholeUD_238 := [[406.26, -32.7, 175.59], [-0.094884, 0.700712, 0.6837, 0.180428], [0,0,0,0], [9E9, 9E9, 9E9, 9E9, 9E9, 9E9]];
	VAR robtarget OpenholeUD_239 := [[402.29, -32.7, 175.07], [-0.106743, 0.699004, 0.680881, 0.19079], [0,0,0,0], [9E9, 9E9, 9E9, 9E9, 9E9, 9E9]];
	VAR robtarget OpenholeUD_240 := [[398.33, -32.7, 174.55], [-0.11828, 0.697144, 0.678003, 0.200777], [0,0,0,0], [9E9, 9E9, 9E9, 9E9, 9E9, 9E9]];
	VAR robtarget OpenholeUD_241 := [[394.36, -32.7, 174.03], [-0.129483, 0.695151, 0.675083, 0.210388], [0,0,0,0], [9E9, 9E9, 9E9, 9E9, 9E9, 9E9]];
	VAR robtarget OpenholeUD_242 := [[389.32, -32.7, 173.36], [-0.143226, 0.692449, 0.671332, 0.222066], [0,0,0,0], [9E9, 9E9, 9E9, 9E9, 9E9, 9E9]];
	VAR robtarget OpenholeUD_243 := [[385.32, -32.7, 173.38], [-0.183051, 0.683002, 0.683002, 0.183051], [0,0,0,0], [9E9, 9E9, 9E9, 9E9, 9E9, 9E9]];
	VAR robtarget OpenholeUD_244 := [[381.32, -32.7, 173.39], [-0.183051, 0.683002, 0.683002, 0.183051], [0,0,0,0], [9E9, 9E9, 9E9, 9E9, 9E9, 9E9]];
	VAR robtarget OpenholeUD_245 := [[377.32, -32.7, 173.4], [-0.183051, 0.683002, 0.683002, 0.183051], [0,0,0,0], [9E9, 9E9, 9E9, 9E9, 9E9, 9E9]];
	VAR robtarget OpenholeUD_246 := [[373.32, -32.7, 173.42], [-0.183051, 0.683002, 0.683002, 0.183051], [0,0,0,0], [9E9, 9E9, 9E9, 9E9, 9E9, 9E9]];
	VAR robtarget OpenholeUD_247 := [[369.32, -32.7, 173.43], [-0.183051, 0.683002, 0.683002, 0.183051], [0,0,0,0], [9E9, 9E9, 9E9, 9E9, 9E9, 9E9]];
	VAR robtarget OpenholeUD_248 := [[369.32, -32.7, 173.43], [-0.183051, 0.683002, 0.683002, 0.183051], [0,0,0,0], [9E9, 9E9, 9E9, 9E9, 9E9, 9E9]];
	VAR robtarget OpenholeUD_249 := [[369.32, -31.5, 174.12], [-0.183051, 0.683002, 0.683002, 0.183051], [0,0,0,0], [9E9, 9E9, 9E9, 9E9, 9E9, 9E9]];
	VAR robtarget OpenholeUD_250 := [[373.32, -31.5, 174.11], [-0.183051, 0.683002, 0.683002, 0.183051], [0,0,0,0], [9E9, 9E9, 9E9, 9E9, 9E9, 9E9]];
	VAR robtarget OpenholeUD_251 := [[377.32, -31.5, 174.1], [-0.183051, 0.683002, 0.683002, 0.183051], [0,0,0,0], [9E9, 9E9, 9E9, 9E9, 9E9, 9E9]];
	VAR robtarget OpenholeUD_252 := [[381.32, -31.5, 174.08], [-0.183051, 0.683002, 0.683002, 0.183051], [0,0,0,0], [9E9, 9E9, 9E9, 9E9, 9E9, 9E9]];
	VAR robtarget OpenholeUD_253 := [[385.32, -31.5, 174.07], [-0.183051, 0.683002, 0.683002, 0.183051], [0,0,0,0], [9E9, 9E9, 9E9, 9E9, 9E9, 9E9]];
	VAR robtarget OpenholeUD_254 := [[389.32, -31.5, 174.06], [-0.146645, 0.691733, 0.672422, 0.218745], [0,0,0,0], [9E9, 9E9, 9E9, 9E9, 9E9, 9E9]];
	VAR robtarget OpenholeUD_255 := [[393.29, -31.5, 174.53], [-0.13593, 0.693919, 0.675351, 0.209527], [0,0,0,0], [9E9, 9E9, 9E9, 9E9, 9E9, 9E9]];
	VAR robtarget OpenholeUD_256 := [[397.27, -31.5, 175.01], [-0.124866, 0.695995, 0.678252, 0.199936], [0,0,0,0], [9E9, 9E9, 9E9, 9E9, 9E9, 9E9]];
	VAR robtarget OpenholeUD_257 := [[401.24, -31.5, 175.49], [-0.113463, 0.697944, 0.68111, 0.18997], [0,0,0,0], [9E9, 9E9, 9E9, 9E9, 9E9, 9E9]];
	VAR robtarget OpenholeUD_258 := [[405.21, -31.5, 175.96], [-0.101731, 0.699751, 0.68391, 0.179629], [0,0,0,0], [9E9, 9E9, 9E9, 9E9, 9E9, 9E9]];
	VAR robtarget OpenholeUD_259 := [[409.18, -31.5, 176.44], [-0.089685, 0.701396, 0.686635, 0.168915], [0,0,0,0], [9E9, 9E9, 9E9, 9E9, 9E9, 9E9]];
	VAR robtarget OpenholeUD_260 := [[413.15, -31.5, 176.92], [-0.077344, 0.702864, 0.689266, 0.157836], [0,0,0,0], [9E9, 9E9, 9E9, 9E9, 9E9, 9E9]];
	VAR robtarget OpenholeUD_261 := [[417.12, -31.5, 177.39], [-0.064733, 0.704138, 0.691785, 0.146401], [0,0,0,0], [9E9, 9E9, 9E9, 9E9, 9E9, 9E9]];
	VAR robtarget OpenholeUD_262 := [[421.1, -31.5, 177.87], [-0.051876, 0.705201, 0.694173, 0.134624], [0,0,0,0], [9E9, 9E9, 9E9, 9E9, 9E9, 9E9]];
	VAR robtarget OpenholeUD_263 := [[425.07, -31.5, 178.35], [-0.038807, 0.706041, 0.696411, 0.122523], [0,0,0,0], [9E9, 9E9, 9E9, 9E9, 9E9, 9E9]];
	VAR robtarget OpenholeUD_264 := [[429.04, -31.5, 178.82], [-0.025559, 0.706645, 0.698479, 0.110122], [0,0,0,0], [9E9, 9E9, 9E9, 9E9, 9E9, 9E9]];
	VAR robtarget OpenholeUD_265 := [[433.01, -31.5, 179.3], [-0.012171, 0.707002, 0.70036, 0.097447], [0,0,0,0], [9E9, 9E9, 9E9, 9E9, 9E9, 9E9]];
	VAR robtarget OpenholeUD_266 := [[436.98, -31.5, 179.78], [0.001316, 0.707106, 0.702036, 0.084529], [0,0,0,0], [9E9, 9E9, 9E9, 9E9, 9E9, 9E9]];
	VAR robtarget OpenholeUD_267 := [[440.95, -31.5, 180.25], [0.014861, 0.706951, 0.703492, 0.071403], [0,0,0,0], [9E9, 9E9, 9E9, 9E9, 9E9, 9E9]];
	VAR robtarget OpenholeUD_268 := [[444.92, -31.5, 180.73], [0.028417, 0.706536, 0.704715, 0.058107], [0,0,0,0], [9E9, 9E9, 9E9, 9E9, 9E9, 9E9]];
	VAR robtarget OpenholeUD_269 := [[448.9, -31.5, 181.21], [0.041941, 0.705862, 0.705694, 0.044682], [0,0,0,0], [9E9, 9E9, 9E9, 9E9, 9E9, 9E9]];
	VAR robtarget OpenholeUD_270 := [[452.87, -31.5, 181.68], [0.055389, 0.704934, 0.706419, 0.031172], [0,0,0,0], [9E9, 9E9, 9E9, 9E9, 9E9, 9E9]];
	VAR robtarget OpenholeUD_271 := [[456.84, -31.5, 182.16], [0.068715, 0.70376, 0.706887, 0.017619], [0,0,0,0], [9E9, 9E9, 9E9, 9E9, 9E9, 9E9]];
	VAR robtarget OpenholeUD_272 := [[460.81, -31.5, 182.64], [0.08188, 0.70235, 0.707095, 0.004071], [0,0,0,0], [9E9, 9E9, 9E9, 9E9, 9E9, 9E9]];
	VAR robtarget OpenholeUD_273 := [[464.78, -31.5, 183.11], [0.094845, 0.700717, 0.707044, -0.009431], [0,0,0,0], [9E9, 9E9, 9E9, 9E9, 9E9, 9E9]];
	VAR robtarget OpenholeUD_274 := [[468.75, -31.5, 183.59], [0.107573, 0.698876, 0.706738, -0.022841], [0,0,0,0], [9E9, 9E9, 9E9, 9E9, 9E9, 9E9]];
	VAR robtarget OpenholeUD_275 := [[472.72, -31.5, 184.07], [0.120034, 0.696844, 0.706184, -0.036119], [0,0,0,0], [9E9, 9E9, 9E9, 9E9, 9E9, 9E9]];
	VAR robtarget OpenholeUD_276 := [[476.7, -31.5, 184.54], [0.132198, 0.694639, 0.705391, -0.049226], [0,0,0,0], [9E9, 9E9, 9E9, 9E9, 9E9, 9E9]];
	VAR robtarget OpenholeUD_277 := [[480.67, -31.5, 185.02], [0.144044, 0.69228, 0.704372, -0.062127], [0,0,0,0], [9E9, 9E9, 9E9, 9E9, 9E9, 9E9]];
	VAR robtarget OpenholeUD_278 := [[484.64, -31.5, 185.5], [0.155551, 0.689785, 0.70314, -0.07479], [0,0,0,0], [9E9, 9E9, 9E9, 9E9, 9E9, 9E9]];
	VAR robtarget OpenholeUD_279 := [[488.61, -31.5, 185.97], [0.166704, 0.687175, 0.701711, -0.087187], [0,0,0,0], [9E9, 9E9, 9E9, 9E9, 9E9, 9E9]];
	VAR robtarget OpenholeUD_280 := [[492.58, -31.5, 186.45], [0.177493, 0.684468, 0.700101, -0.099294], [0,0,0,0], [9E9, 9E9, 9E9, 9E9, 9E9, 9E9]];
	VAR robtarget OpenholeUD_281 := [[496.55, -31.5, 186.93], [0.187911, 0.681681, 0.698326, -0.11109], [0,0,0,0], [9E9, 9E9, 9E9, 9E9, 9E9, 9E9]];
	VAR robtarget OpenholeUD_282 := [[500.53, -31.5, 187.4], [0.197953, 0.678833, 0.696404, -0.122561], [0,0,0,0], [9E9, 9E9, 9E9, 9E9, 9E9, 9E9]];
	VAR robtarget OpenholeUD_283 := [[504.5, -31.5, 187.88], [0.20762, 0.675939, 0.694353, -0.133694], [0,0,0,0], [9E9, 9E9, 9E9, 9E9, 9E9, 9E9]];
	VAR robtarget OpenholeUD_284 := [[509.37, -31.5, 188.46], [0.183051, 0.683002, 0.683002, -0.183051], [0,0,0,0], [9E9, 9E9, 9E9, 9E9, 9E9, 9E9]];
	VAR robtarget OpenholeUD_285 := [[513.37, -31.5, 188.45], [0.183051, 0.683002, 0.683002, -0.183051], [0,0,0,0], [9E9, 9E9, 9E9, 9E9, 9E9, 9E9]];
	VAR robtarget OpenholeUD_286 := [[517.37, -31.5, 188.44], [0.183051, 0.683002, 0.683002, -0.183051], [0,0,0,0], [9E9, 9E9, 9E9, 9E9, 9E9, 9E9]];
	VAR robtarget OpenholeUD_287 := [[521.37, -31.5, 188.43], [0.183051, 0.683002, 0.683002, -0.183051], [0,0,0,0], [9E9, 9E9, 9E9, 9E9, 9E9, 9E9]];
	VAR robtarget OpenholeUD_288 := [[525.37, -31.5, 188.41], [0.183051, 0.683002, 0.683002, -0.183051], [0,0,0,0], [9E9, 9E9, 9E9, 9E9, 9E9, 9E9]];
	VAR robtarget OpenholeUD_289 := [[529.37, -31.5, 188.4], [0.183051, 0.683002, 0.683002, -0.183051], [0,0,0,0], [9E9, 9E9, 9E9, 9E9, 9E9, 9E9]];
	VAR robtarget OpenholeUD_290 := [[529.37, -31.5, 188.4], [0.183051, 0.683002, 0.683002, -0.183051], [0,0,0,0], [9E9, 9E9, 9E9, 9E9, 9E9, 9E9]];
	VAR robtarget OpenholeUD_291 := [[529.37, -30.3, 187.71], [0.183051, 0.683002, 0.683002, -0.183051], [0,0,0,0], [9E9, 9E9, 9E9, 9E9, 9E9, 9E9]];
	VAR robtarget OpenholeUD_292 := [[525.37, -30.3, 187.72], [0.183051, 0.683002, 0.683002, -0.183051], [0,0,0,0], [9E9, 9E9, 9E9, 9E9, 9E9, 9E9]];
	VAR robtarget OpenholeUD_293 := [[521.37, -30.3, 187.73], [0.183051, 0.683002, 0.683002, -0.183051], [0,0,0,0], [9E9, 9E9, 9E9, 9E9, 9E9, 9E9]];
	VAR robtarget OpenholeUD_294 := [[517.37, -30.3, 187.75], [0.183051, 0.683002, 0.683002, -0.183051], [0,0,0,0], [9E9, 9E9, 9E9, 9E9, 9E9, 9E9]];
	VAR robtarget OpenholeUD_295 := [[513.37, -30.3, 187.76], [0.183051, 0.683002, 0.683002, -0.183051], [0,0,0,0], [9E9, 9E9, 9E9, 9E9, 9E9, 9E9]];
	VAR robtarget OpenholeUD_296 := [[509.37, -30.3, 187.77], [0.183051, 0.683002, 0.683002, -0.183051], [0,0,0,0], [9E9, 9E9, 9E9, 9E9, 9E9, 9E9]];
	VAR robtarget OpenholeUD_297 := [[505.39, -30.3, 187.34], [0.206349, 0.676328, 0.693181, -0.139642], [0,0,0,0], [9E9, 9E9, 9E9, 9E9, 9E9, 9E9]];
	VAR robtarget OpenholeUD_298 := [[501.41, -30.3, 186.91], [0.196687, 0.679201, 0.695308, -0.128636], [0,0,0,0], [9E9, 9E9, 9E9, 9E9, 9E9, 9E9]];
	VAR robtarget OpenholeUD_299 := [[497.44, -30.3, 186.48], [0.186649, 0.682028, 0.697312, -0.117288], [0,0,0,0], [9E9, 9E9, 9E9, 9E9, 9E9, 9E9]];
	VAR robtarget OpenholeUD_300 := [[493.46, -30.3, 186.05], [0.176237, 0.684792, 0.699176, -0.105607], [0,0,0,0], [9E9, 9E9, 9E9, 9E9, 9E9, 9E9]];
	VAR robtarget OpenholeUD_301 := [[489.48, -30.3, 185.62], [0.165454, 0.687477, 0.700883, -0.093608], [0,0,0,0], [9E9, 9E9, 9E9, 9E9, 9E9, 9E9]];
	VAR robtarget OpenholeUD_302 := [[485.51, -30.3, 185.18], [0.154306, 0.690065, 0.702416, -0.081311], [0,0,0,0], [9E9, 9E9, 9E9, 9E9, 9E9, 9E9]];
	VAR robtarget OpenholeUD_303 := [[481.53, -30.3, 184.75], [0.142805, 0.692536, 0.703758, -0.068736], [0,0,0,0], [9E9, 9E9, 9E9, 9E9, 9E9, 9E9]];
	VAR robtarget OpenholeUD_304 := [[477.55, -30.3, 184.32], [0.130965, 0.694873, 0.704893, -0.055912], [0,0,0,0], [9E9, 9E9, 9E9, 9E9, 9E9, 9E9]];
	VAR robtarget OpenholeUD_305 := [[473.58, -30.3, 183.89], [0.118805, 0.697055, 0.705806, -0.042868], [0,0,0,0], [9E9, 9E9, 9E9, 9E9, 9E9, 9E9]];
	VAR robtarget OpenholeUD_306 := [[469.6, -30.3, 183.46], [0.106348, 0.699064, 0.706485, -0.029639], [0,0,0,0], [9E9, 9E9, 9E9, 9E9, 9E9, 9E9]];
	VAR robtarget OpenholeUD_307 := [[465.62, -30.3, 183.03], [0.093622, 0.700882, 0.70692, -0.016263], [0,0,0,0], [9E9, 9E9, 9E9, 9E9, 9E9, 9E9]];
	VAR robtarget OpenholeUD_308 := [[461.65, -30.3, 182.6], [0.080658, 0.702492, 0.707101, -0.002781], [0,0,0,0], [9E9, 9E9, 9E9, 9E9, 9E9, 9E9]];
	VAR robtarget OpenholeUD_309 := [[457.67, -30.3, 182.16], [0.067491, 0.703878, 0.707025, 0.010766], [0,0,0,0], [9E9, 9E9, 9E9, 9E9, 9E9, 9E9]];
	VAR robtarget OpenholeUD_310 := [[453.69, -30.3, 181.73], [0.054161, 0.705029, 0.706688, 0.024332], [0,0,0,0], [9E9, 9E9, 9E9, 9E9, 9E9, 9E9]];
	VAR robtarget OpenholeUD_311 := [[449.72, -30.3, 181.3], [0.040709, 0.705934, 0.706092, 0.037873], [0,0,0,0], [9E9, 9E9, 9E9, 9E9, 9E9, 9E9]];
	VAR robtarget OpenholeUD_312 := [[445.74, -30.3, 180.87], [0.027177, 0.706584, 0.70524, 0.051344], [0,0,0,0], [9E9, 9E9, 9E9, 9E9, 9E9, 9E9]];
	VAR robtarget OpenholeUD_313 := [[441.76, -30.3, 180.44], [0.01361, 0.706976, 0.70414, 0.064702], [0,0,0,0], [9E9, 9E9, 9E9, 9E9, 9E9, 9E9]];
	VAR robtarget OpenholeUD_314 := [[437.79, -30.3, 180.01], [0.000054, 0.707107, 0.702802, 0.077905], [0,0,0,0], [9E9, 9E9, 9E9, 9E9, 9E9, 9E9]];
	VAR robtarget OpenholeUD_315 := [[433.81, -30.3, 179.58], [-0.013447, 0.706979, 0.701238, 0.090913], [0,0,0,0], [9E9, 9E9, 9E9, 9E9, 9E9, 9E9]];
	VAR robtarget OpenholeUD_316 := [[429.83, -30.3, 179.14], [-0.02685, 0.706597, 0.699463, 0.10369], [0,0,0,0], [9E9, 9E9, 9E9, 9E9, 9E9, 9E9]];
	VAR robtarget OpenholeUD_317 := [[425.86, -30.3, 178.71], [-0.040114, 0.705968, 0.697493, 0.116205], [0,0,0,0], [9E9, 9E9, 9E9, 9E9, 9E9, 9E9]];
	VAR robtarget OpenholeUD_318 := [[421.88, -30.3, 178.28], [-0.053201, 0.705103, 0.695346, 0.128428], [0,0,0,0], [9E9, 9E9, 9E9, 9E9, 9E9, 9E9]];
	VAR robtarget OpenholeUD_319 := [[417.9, -30.3, 177.85], [-0.066075, 0.704013, 0.693041, 0.140336], [0,0,0,0], [9E9, 9E9, 9E9, 9E9, 9E9, 9E9]];
	VAR robtarget OpenholeUD_320 := [[413.93, -30.3, 177.42], [-0.078706, 0.702713, 0.690597, 0.151909], [0,0,0,0], [9E9, 9E9, 9E9, 9E9, 9E9, 9E9]];
	VAR robtarget OpenholeUD_321 := [[409.95, -30.3, 176.99], [-0.091065, 0.701218, 0.688032, 0.163131], [0,0,0,0], [9E9, 9E9, 9E9, 9E9, 9E9, 9E9]];
	VAR robtarget OpenholeUD_322 := [[405.97, -30.3, 176.56], [-0.103129, 0.699546, 0.685366, 0.173991], [0,0,0,0], [9E9, 9E9, 9E9, 9E9, 9E9, 9E9]];
	VAR robtarget OpenholeUD_323 := [[402, -30.3, 176.13], [-0.114878, 0.697713, 0.682618, 0.184481], [0,0,0,0], [9E9, 9E9, 9E9, 9E9, 9E9, 9E9]];
	VAR robtarget OpenholeUD_324 := [[398.02, -30.3, 175.69], [-0.126298, 0.695736, 0.679803, 0.194597], [0,0,0,0], [9E9, 9E9, 9E9, 9E9, 9E9, 9E9]];
	VAR robtarget OpenholeUD_325 := [[394.04, -30.3, 175.26], [-0.137377, 0.693634, 0.676939, 0.204338], [0,0,0,0], [9E9, 9E9, 9E9, 9E9, 9E9, 9E9]];
	VAR robtarget OpenholeUD_326 := [[389.33, -30.3, 174.75], [-0.150067, 0.690999, 0.673497, 0.215411], [0,0,0,0], [9E9, 9E9, 9E9, 9E9, 9E9, 9E9]];
	VAR robtarget OpenholeUD_327 := [[385.33, -30.3, 174.76], [-0.183051, 0.683002, 0.683002, 0.183051], [0,0,0,0], [9E9, 9E9, 9E9, 9E9, 9E9, 9E9]];
	VAR robtarget OpenholeUD_328 := [[381.33, -30.3, 174.78], [-0.183051, 0.683002, 0.683002, 0.183051], [0,0,0,0], [9E9, 9E9, 9E9, 9E9, 9E9, 9E9]];
	VAR robtarget OpenholeUD_329 := [[377.33, -30.3, 174.79], [-0.183051, 0.683002, 0.683002, 0.183051], [0,0,0,0], [9E9, 9E9, 9E9, 9E9, 9E9, 9E9]];
	VAR robtarget OpenholeUD_330 := [[373.33, -30.3, 174.8], [-0.183051, 0.683002, 0.683002, 0.183051], [0,0,0,0], [9E9, 9E9, 9E9, 9E9, 9E9, 9E9]];
	VAR robtarget OpenholeUD_331 := [[369.33, -30.3, 174.81], [-0.183051, 0.683002, 0.683002, 0.183051], [0,0,0,0], [9E9, 9E9, 9E9, 9E9, 9E9, 9E9]];
	VAR robtarget OpenholeUD_332 := [[369.33, -30.3, 174.81], [-0.183051, 0.683002, 0.683002, 0.183051], [0,0,0,0], [9E9, 9E9, 9E9, 9E9, 9E9, 9E9]];
	VAR robtarget OpenholeUD_333 := [[369.33, -29.1, 175.51], [-0.183051, 0.683002, 0.683002, 0.183051], [0,0,0,0], [9E9, 9E9, 9E9, 9E9, 9E9, 9E9]];
	VAR robtarget OpenholeUD_334 := [[373.33, -29.1, 175.49], [-0.183051, 0.683002, 0.683002, 0.183051], [0,0,0,0], [9E9, 9E9, 9E9, 9E9, 9E9, 9E9]];
	VAR robtarget OpenholeUD_335 := [[377.33, -29.1, 175.48], [-0.183051, 0.683002, 0.683002, 0.183051], [0,0,0,0], [9E9, 9E9, 9E9, 9E9, 9E9, 9E9]];
	VAR robtarget OpenholeUD_336 := [[381.33, -29.1, 175.47], [-0.183051, 0.683002, 0.683002, 0.183051], [0,0,0,0], [9E9, 9E9, 9E9, 9E9, 9E9, 9E9]];
	VAR robtarget OpenholeUD_337 := [[385.33, -29.1, 175.46], [-0.183051, 0.683002, 0.683002, 0.183051], [0,0,0,0], [9E9, 9E9, 9E9, 9E9, 9E9, 9E9]];
	VAR robtarget OpenholeUD_338 := [[389.33, -29.1, 175.44], [-0.153493, 0.690246, 0.674558, 0.212066], [0,0,0,0], [9E9, 9E9, 9E9, 9E9, 9E9, 9E9]];
	VAR robtarget OpenholeUD_339 := [[393.31, -29.1, 175.83], [-0.142882, 0.69252, 0.677435, 0.202687], [0,0,0,0], [9E9, 9E9, 9E9, 9E9, 9E9, 9E9]];
	VAR robtarget OpenholeUD_340 := [[397.29, -29.1, 176.22], [-0.13192, 0.694692, 0.680276, 0.192936], [0,0,0,0], [9E9, 9E9, 9E9, 9E9, 9E9, 9E9]];
	VAR robtarget OpenholeUD_341 := [[401.27, -29.1, 176.6], [-0.120611, 0.696745, 0.683067, 0.182811], [0,0,0,0], [9E9, 9E9, 9E9, 9E9, 9E9, 9E9]];
	VAR robtarget OpenholeUD_342 := [[405.25, -29.1, 176.99], [-0.108967, 0.69866, 0.68579, 0.172312], [0,0,0,0], [9E9, 9E9, 9E9, 9E9, 9E9, 9E9]];
	VAR robtarget OpenholeUD_343 := [[409.23, -29.1, 177.37], [-0.097002, 0.700422, 0.68843, 0.161444], [0,0,0,0], [9E9, 9E9, 9E9, 9E9, 9E9, 9E9]];
	VAR robtarget OpenholeUD_344 := [[413.22, -29.1, 177.76], [-0.084734, 0.702011, 0.690967, 0.150214], [0,0,0,0], [9E9, 9E9, 9E9, 9E9, 9E9, 9E9]];
	VAR robtarget OpenholeUD_345 := [[417.2, -29.1, 178.15], [-0.072185, 0.703413, 0.693383, 0.138634], [0,0,0,0], [9E9, 9E9, 9E9, 9E9, 9E9, 9E9]];
	VAR robtarget OpenholeUD_346 := [[421.18, -29.1, 178.53], [-0.059381, 0.704609, 0.69566, 0.12672], [0,0,0,0], [9E9, 9E9, 9E9, 9E9, 9E9, 9E9]];
	VAR robtarget OpenholeUD_347 := [[425.16, -29.1, 178.92], [-0.046354, 0.705586, 0.697777, 0.114489], [0,0,0,0], [9E9, 9E9, 9E9, 9E9, 9E9, 9E9]];
	VAR robtarget OpenholeUD_348 := [[429.14, -29.1, 179.3], [-0.033136, 0.70633, 0.699716, 0.101968], [0,0,0,0], [9E9, 9E9, 9E9, 9E9, 9E9, 9E9]];
	VAR robtarget OpenholeUD_349 := [[433.12, -29.1, 179.69], [-0.019765, 0.70683, 0.70146, 0.089184], [0,0,0,0], [9E9, 9E9, 9E9, 9E9, 9E9, 9E9]];
	VAR robtarget OpenholeUD_350 := [[437.1, -29.1, 180.07], [-0.006283, 0.707079, 0.702992, 0.076169], [0,0,0,0], [9E9, 9E9, 9E9, 9E9, 9E9, 9E9]];
	VAR robtarget OpenholeUD_351 := [[441.08, -29.1, 180.46], [0.007269, 0.707069, 0.704298, 0.062959], [0,0,0,0], [9E9, 9E9, 9E9, 9E9, 9E9, 9E9]];
	VAR robtarget OpenholeUD_352 := [[445.07, -29.1, 180.85], [0.020846, 0.706799, 0.705366, 0.049593], [0,0,0,0], [9E9, 9E9, 9E9, 9E9, 9E9, 9E9]];
	VAR robtarget OpenholeUD_353 := [[449.05, -29.1, 181.23], [0.034403, 0.706269, 0.706184, 0.036114], [0,0,0,0], [9E9, 9E9, 9E9, 9E9, 9E9, 9E9]];
	VAR robtarget OpenholeUD_354 := [[453.03, -29.1, 181.62], [0.047896, 0.705483, 0.706747, 0.022564], [0,0,0,0], [9E9, 9E9, 9E9, 9E9, 9E9, 9E9]];
	VAR robtarget OpenholeUD_355 := [[457.01, -29.1, 182], [0.06128, 0.704446, 0.70705, 0.008989], [0,0,0,0], [9E9, 9E9, 9E9, 9E9, 9E9, 9E9]];
	VAR robtarget OpenholeUD_356 := [[460.99, -29.1, 182.39], [0.074513, 0.70317, 0.707092, -0.004567], [0,0,0,0], [9E9, 9E9, 9E9, 9E9, 9E9, 9E9]];
	VAR robtarget OpenholeUD_357 := [[464.97, -29.1, 182.78], [0.087557, 0.701665, 0.706876, -0.018059], [0,0,0,0], [9E9, 9E9, 9E9, 9E9, 9E9, 9E9]];
	VAR robtarget OpenholeUD_358 := [[468.95, -29.1, 183.16], [0.100374, 0.699947, 0.706407, -0.031444], [0,0,0,0], [9E9, 9E9, 9E9, 9E9, 9E9, 9E9]];
	VAR robtarget OpenholeUD_359 := [[472.94, -29.1, 183.55], [0.112931, 0.69803, 0.705694, -0.044682], [0,0,0,0], [9E9, 9E9, 9E9, 9E9, 9E9, 9E9]];
	VAR robtarget OpenholeUD_360 := [[476.92, -29.1, 183.93], [0.125201, 0.695934, 0.704746, -0.057734], [0,0,0,0], [9E9, 9E9, 9E9, 9E9, 9E9, 9E9]];
	VAR robtarget OpenholeUD_361 := [[480.9, -29.1, 184.32], [0.137158, 0.693677, 0.703577, -0.070567], [0,0,0,0], [9E9, 9E9, 9E9, 9E9, 9E9, 9E9]];
	VAR robtarget OpenholeUD_362 := [[484.88, -29.1, 184.71], [0.148782, 0.691277, 0.702201, -0.083148], [0,0,0,0], [9E9, 9E9, 9E9, 9E9, 9E9, 9E9]];
	VAR robtarget OpenholeUD_363 := [[488.86, -29.1, 185.09], [0.160057, 0.688754, 0.700635, -0.095452], [0,0,0,0], [9E9, 9E9, 9E9, 9E9, 9E9, 9E9]];
	VAR robtarget OpenholeUD_364 := [[492.84, -29.1, 185.48], [0.170972, 0.686126, 0.698894, -0.107456], [0,0,0,0], [9E9, 9E9, 9E9, 9E9, 9E9, 9E9]];
	VAR robtarget OpenholeUD_365 := [[496.82, -29.1, 185.86], [0.181518, 0.683411, 0.696998, -0.119141], [0,0,0,0], [9E9, 9E9, 9E9, 9E9, 9E9, 9E9]];
	VAR robtarget OpenholeUD_366 := [[500.81, -29.1, 186.25], [0.191691, 0.680628, 0.694962, -0.130491], [0,0,0,0], [9E9, 9E9, 9E9, 9E9, 9E9, 9E9]];
	VAR robtarget OpenholeUD_367 := [[504.79, -29.1, 186.64], [0.20149, 0.677792, 0.692805, -0.141498], [0,0,0,0], [9E9, 9E9, 9E9, 9E9, 9E9, 9E9]];
	VAR robtarget OpenholeUD_368 := [[509.36, -29.1, 187.08], [0.183051, 0.683002, 0.683002, -0.183051], [0,0,0,0], [9E9, 9E9, 9E9, 9E9, 9E9, 9E9]];
	VAR robtarget OpenholeUD_369 := [[513.36, -29.1, 187.07], [0.183051, 0.683002, 0.683002, -0.183051], [0,0,0,0], [9E9, 9E9, 9E9, 9E9, 9E9, 9E9]];
	VAR robtarget OpenholeUD_370 := [[517.36, -29.1, 187.05], [0.183051, 0.683002, 0.683002, -0.183051], [0,0,0,0], [9E9, 9E9, 9E9, 9E9, 9E9, 9E9]];
	VAR robtarget OpenholeUD_371 := [[521.36, -29.1, 187.04], [0.183051, 0.683002, 0.683002, -0.183051], [0,0,0,0], [9E9, 9E9, 9E9, 9E9, 9E9, 9E9]];
	VAR robtarget OpenholeUD_372 := [[529.36, -29.1, 187.02], [0.183051, 0.683002, 0.683002, -0.183051], [0,0,0,0], [9E9, 9E9, 9E9, 9E9, 9E9, 9E9]];
	VAR robtarget OpenholeUD_373 := [[529.36, -29.1, 187.02], [0.183051, 0.683002, 0.683002, -0.183051], [0,0,0,0], [9E9, 9E9, 9E9, 9E9, 9E9, 9E9]];
	VAR robtarget OpenholeUD_374 := [[529.36, -27.9, 186.32], [0.183051, 0.683002, 0.683002, -0.183051], [0,0,0,0], [9E9, 9E9, 9E9, 9E9, 9E9, 9E9]];
	VAR robtarget OpenholeUD_375 := [[525.36, -27.9, 186.34], [0.183051, 0.683002, 0.683002, -0.183051], [0,0,0,0], [9E9, 9E9, 9E9, 9E9, 9E9, 9E9]];
	VAR robtarget OpenholeUD_376 := [[521.36, -27.9, 186.35], [0.183051, 0.683002, 0.683002, -0.183051], [0,0,0,0], [9E9, 9E9, 9E9, 9E9, 9E9, 9E9]];
	VAR robtarget OpenholeUD_377 := [[517.36, -27.9, 186.36], [0.183051, 0.683002, 0.683002, -0.183051], [0,0,0,0], [9E9, 9E9, 9E9, 9E9, 9E9, 9E9]];
	VAR robtarget OpenholeUD_378 := [[509.36, -27.9, 186.39], [0.183051, 0.683002, 0.683002, -0.183051], [0,0,0,0], [9E9, 9E9, 9E9, 9E9, 9E9, 9E9]];
	VAR robtarget OpenholeUD_379 := [[505.38, -27.9, 186.05], [0.199494, 0.678382, 0.691743, -0.146598], [0,0,0,0], [9E9, 9E9, 9E9, 9E9, 9E9, 9E9]];
	VAR robtarget OpenholeUD_380 := [[501.39, -27.9, 185.71], [0.189673, 0.681193, 0.693964, -0.135697], [0,0,0,0], [9E9, 9E9, 9E9, 9E9, 9E9, 9E9]];
	VAR robtarget OpenholeUD_381 := [[497.41, -27.9, 185.37], [0.179478, 0.68395, 0.696069, -0.124448], [0,0,0,0], [9E9, 9E9, 9E9, 9E9, 9E9, 9E9]];
	VAR robtarget OpenholeUD_382 := [[493.42, -27.9, 185.02], [0.16891, 0.686636, 0.698042, -0.112861], [0,0,0,0], [9E9, 9E9, 9E9, 9E9, 9E9, 9E9]];
	VAR robtarget OpenholeUD_383 := [[489.43, -27.9, 184.68], [0.157975, 0.689234, 0.699864, -0.100948], [0,0,0,0], [9E9, 9E9, 9E9, 9E9, 9E9, 9E9]];
	VAR robtarget OpenholeUD_384 := [[485.45, -27.9, 184.34], [0.14668, 0.691726, 0.701518, -0.088728], [0,0,0,0], [9E9, 9E9, 9E9, 9E9, 9E9, 9E9]];
	VAR robtarget OpenholeUD_385 := [[481.46, -27.9, 184], [0.135037, 0.694093, 0.702987, -0.076221], [0,0,0,0], [9E9, 9E9, 9E9, 9E9, 9E9, 9E9]];
	VAR robtarget OpenholeUD_386 := [[477.48, -27.9, 183.66], [0.123062, 0.696316, 0.704254, -0.063455], [0,0,0,0], [9E9, 9E9, 9E9, 9E9, 9E9, 9E9]];
	VAR robtarget OpenholeUD_387 := [[473.49, -27.9, 183.32], [0.110776, 0.698376, 0.705304, -0.050458], [0,0,0,0], [9E9, 9E9, 9E9, 9E9, 9E9, 9E9]];
	VAR robtarget OpenholeUD_388 := [[469.51, -27.9, 182.98], [0.098203, 0.700254, 0.706124, -0.037264], [0,0,0,0], [9E9, 9E9, 9E9, 9E9, 9E9, 9E9]];
	VAR robtarget OpenholeUD_389 := [[465.52, -27.9, 182.64], [0.085371, 0.701934, 0.706702, -0.023911], [0,0,0,0], [9E9, 9E9, 9E9, 9E9, 9E9, 9E9]];
	VAR robtarget OpenholeUD_390 := [[461.54, -27.9, 182.3], [0.072314, 0.703399, 0.70703, -0.010439], [0,0,0,0], [9E9, 9E9, 9E9, 9E9, 9E9, 9E9]];
	VAR robtarget OpenholeUD_391 := [[457.55, -27.9, 181.96], [0.059068, 0.704635, 0.7071, 0.00311], [0,0,0,0], [9E9, 9E9, 9E9, 9E9, 9E9, 9E9]];
	VAR robtarget OpenholeUD_392 := [[453.57, -27.9, 181.62], [0.045672, 0.70563, 0.70691, 0.016692], [0,0,0,0], [9E9, 9E9, 9E9, 9E9, 9E9, 9E9]];
	VAR robtarget OpenholeUD_393 := [[449.58, -27.9, 181.28], [0.032169, 0.706375, 0.706459, 0.030262], [0,0,0,0], [9E9, 9E9, 9E9, 9E9, 9E9, 9E9]];
	VAR robtarget OpenholeUD_394 := [[445.59, -27.9, 180.94], [0.018603, 0.706862, 0.705751, 0.043774], [0,0,0,0], [9E9, 9E9, 9E9, 9E9, 9E9, 9E9]];
	VAR robtarget OpenholeUD_395 := [[441.61, -27.9, 180.6], [0.005018, 0.707089, 0.704791, 0.057186], [0,0,0,0], [9E9, 9E9, 9E9, 9E9, 9E9, 9E9]];
	VAR robtarget OpenholeUD_396 := [[437.62, -27.9, 180.26], [-0.00854, 0.707055, 0.703588, 0.070454], [0,0,0,0], [9E9, 9E9, 9E9, 9E9, 9E9, 9E9]];
	VAR robtarget OpenholeUD_397 := [[433.64, -27.9, 179.92], [-0.022028, 0.706764, 0.702155, 0.083538], [0,0,0,0], [9E9, 9E9, 9E9, 9E9, 9E9, 9E9]];
	VAR robtarget OpenholeUD_398 := [[429.65, -27.9, 179.58], [-0.035402, 0.70622, 0.700505, 0.096402], [0,0,0,0], [9E9, 9E9, 9E9, 9E9, 9E9, 9E9]];
	VAR robtarget OpenholeUD_399 := [[425.67, -27.9, 179.24], [-0.048622, 0.705433, 0.698653, 0.109012], [0,0,0,0], [9E9, 9E9, 9E9, 9E9, 9E9, 9E9]];
	VAR robtarget OpenholeUD_400 := [[421.68, -27.9, 178.9], [-0.06165, 0.704414, 0.696618, 0.121339], [0,0,0,0], [9E9, 9E9, 9E9, 9E9, 9E9, 9E9]];
	VAR robtarget OpenholeUD_401 := [[417.7, -27.9, 178.56], [-0.074452, 0.703176, 0.694418, 0.133358], [0,0,0,0], [9E9, 9E9, 9E9, 9E9, 9E9, 9E9]];
	VAR robtarget OpenholeUD_402 := [[413.71, -27.9, 178.22], [-0.086998, 0.701735, 0.69207, 0.145047], [0,0,0,0], [9E9, 9E9, 9E9, 9E9, 9E9, 9E9]];
	VAR robtarget OpenholeUD_403 := [[409.72, -27.9, 177.88], [-0.099261, 0.700105, 0.689595, 0.156391], [0,0,0,0], [9E9, 9E9, 9E9, 9E9, 9E9, 9E9]];
	VAR robtarget OpenholeUD_404 := [[405.74, -27.9, 177.54], [-0.111219, 0.698305, 0.687012, 0.167377], [0,0,0,0], [9E9, 9E9, 9E9, 9E9, 9E9, 9E9]];
	VAR robtarget OpenholeUD_405 := [[401.75, -27.9, 177.2], [-0.122855, 0.696352, 0.684337, 0.177996], [0,0,0,0], [9E9, 9E9, 9E9, 9E9, 9E9, 9E9]];
	VAR robtarget OpenholeUD_406 := [[397.77, -27.9, 176.86], [-0.134153, 0.694264, 0.68159, 0.188243], [0,0,0,0], [9E9, 9E9, 9E9, 9E9, 9E9, 9E9]];
	VAR robtarget OpenholeUD_407 := [[393.78, -27.9, 176.52], [-0.145103, 0.692059, 0.678785, 0.198117], [0,0,0,0], [9E9, 9E9, 9E9, 9E9, 9E9, 9E9]];
	VAR robtarget OpenholeUD_408 := [[389.33, -27.9, 176.14], [-0.15692, 0.689475, 0.675604, 0.208709], [0,0,0,0], [9E9, 9E9, 9E9, 9E9, 9E9, 9E9]];
	VAR robtarget OpenholeUD_409 := [[385.33, -27.9, 176.15], [-0.183051, 0.683002, 0.683002, 0.183051], [0,0,0,0], [9E9, 9E9, 9E9, 9E9, 9E9, 9E9]];
	VAR robtarget OpenholeUD_410 := [[381.33, -27.9, 176.16], [-0.183051, 0.683002, 0.683002, 0.183051], [0,0,0,0], [9E9, 9E9, 9E9, 9E9, 9E9, 9E9]];
	VAR robtarget OpenholeUD_411 := [[377.33, -27.9, 176.17], [-0.183051, 0.683002, 0.683002, 0.183051], [0,0,0,0], [9E9, 9E9, 9E9, 9E9, 9E9, 9E9]];
	VAR robtarget OpenholeUD_412 := [[369.33, -27.9, 176.2], [-0.183051, 0.683002, 0.683002, 0.183051], [0,0,0,0], [9E9, 9E9, 9E9, 9E9, 9E9, 9E9]];
	VAR robtarget OpenholeUD_413 := [[369.33, -27.9, 176.2], [-0.183051, 0.683002, 0.683002, 0.183051], [0,0,0,0], [9E9, 9E9, 9E9, 9E9, 9E9, 9E9]];
	VAR robtarget OpenholeUD_414 := [[369.33, -26.7, 176.89], [-0.183051, 0.683002, 0.683002, 0.183051], [0,0,0,0], [9E9, 9E9, 9E9, 9E9, 9E9, 9E9]];
	VAR robtarget OpenholeUD_415 := [[373.33, -26.7, 176.88], [-0.183051, 0.683002, 0.683002, 0.183051], [0,0,0,0], [9E9, 9E9, 9E9, 9E9, 9E9, 9E9]];
	VAR robtarget OpenholeUD_416 := [[377.33, -26.7, 176.87], [-0.183051, 0.683002, 0.683002, 0.183051], [0,0,0,0], [9E9, 9E9, 9E9, 9E9, 9E9, 9E9]];
	VAR robtarget OpenholeUD_417 := [[381.33, -26.7, 176.86], [-0.183051, 0.683002, 0.683002, 0.183051], [0,0,0,0], [9E9, 9E9, 9E9, 9E9, 9E9, 9E9]];
	VAR robtarget OpenholeUD_418 := [[385.33, -26.7, 176.84], [-0.183051, 0.683002, 0.683002, 0.183051], [0,0,0,0], [9E9, 9E9, 9E9, 9E9, 9E9, 9E9]];
	VAR robtarget OpenholeUD_419 := [[389.33, -26.7, 176.83], [-0.160348, 0.688686, 0.676635, 0.205343], [0,0,0,0], [9E9, 9E9, 9E9, 9E9, 9E9, 9E9]];
	VAR robtarget OpenholeUD_420 := [[393.32, -26.7, 177.12], [-0.149852, 0.691046, 0.679455, 0.195807], [0,0,0,0], [9E9, 9E9, 9E9, 9E9, 9E9, 9E9]];
	VAR robtarget OpenholeUD_421 := [[397.31, -26.7, 177.42], [-0.138998, 0.693311, 0.682233, 0.185899], [0,0,0,0], [9E9, 9E9, 9E9, 9E9, 9E9, 9E9]];
	VAR robtarget OpenholeUD_422 := [[401.3, -26.7, 177.71], [-0.127793, 0.695463, 0.684951, 0.175619], [0,0,0,0], [9E9, 9E9, 9E9, 9E9, 9E9, 9E9]];
	VAR robtarget OpenholeUD_423 := [[405.29, -26.7, 178.01], [-0.116247, 0.697486, 0.687594, 0.164967], [0,0,0,0], [9E9, 9E9, 9E9, 9E9, 9E9, 9E9]];
	VAR robtarget OpenholeUD_424 := [[409.28, -26.7, 178.3], [-0.104372, 0.699361, 0.690144, 0.153951], [0,0,0,0], [9E9, 9E9, 9E9, 9E9, 9E9, 9E9]];
	VAR robtarget OpenholeUD_425 := [[413.27, -26.7, 178.6], [-0.092186, 0.701072, 0.692583, 0.142577], [0,0,0,0], [9E9, 9E9, 9E9, 9E9, 9E9, 9E9]];
	VAR robtarget OpenholeUD_426 := [[417.26, -26.7, 178.89], [-0.079709, 0.7026, 0.694893, 0.130859], [0,0,0,0], [9E9, 9E9, 9E9, 9E9, 9E9, 9E9]];
	VAR robtarget OpenholeUD_427 := [[421.24, -26.7, 179.19], [-0.066968, 0.703928, 0.697053, 0.118813], [0,0,0,0], [9E9, 9E9, 9E9, 9E9, 9E9, 9E9]];
	VAR robtarget OpenholeUD_428 := [[425.23, -26.7, 179.48], [-0.053992, 0.705042, 0.699046, 0.106461], [0,0,0,0], [9E9, 9E9, 9E9, 9E9, 9E9, 9E9]];
	VAR robtarget OpenholeUD_429 := [[429.22, -26.7, 179.78], [-0.040814, 0.705928, 0.700854, 0.093828], [0,0,0,0], [9E9, 9E9, 9E9, 9E9, 9E9, 9E9]];
	VAR robtarget OpenholeUD_430 := [[433.21, -26.7, 180.07], [-0.027471, 0.706573, 0.702459, 0.080944], [0,0,0,0], [9E9, 9E9, 9E9, 9E9, 9E9, 9E9]];
	VAR robtarget OpenholeUD_431 := [[437.2, -26.7, 180.36], [-0.014003, 0.706968, 0.703845, 0.06784], [0,0,0,0], [9E9, 9E9, 9E9, 9E9, 9E9, 9E9]];
	VAR robtarget OpenholeUD_432 := [[441.19, -26.7, 180.66], [-0.000452, 0.707107, 0.704999, 0.054556], [0,0,0,0], [9E9, 9E9, 9E9, 9E9, 9E9, 9E9]];
	VAR robtarget OpenholeUD_433 := [[445.18, -26.7, 180.95], [0.013137, 0.706985, 0.70591, 0.041131], [0,0,0,0], [9E9, 9E9, 9E9, 9E9, 9E9, 9E9]];
	VAR robtarget OpenholeUD_434 := [[449.17, -26.7, 181.25], [0.02672, 0.706602, 0.706568, 0.027607], [0,0,0,0], [9E9, 9E9, 9E9, 9E9, 9E9, 9E9]];
	VAR robtarget OpenholeUD_435 := [[453.16, -26.7, 181.54], [0.040251, 0.70596, 0.706968, 0.014028], [0,0,0,0], [9E9, 9E9, 9E9, 9E9, 9E9, 9E9]];
	VAR robtarget OpenholeUD_436 := [[457.15, -26.7, 181.84], [0.053686, 0.705066, 0.707107, 0.00044], [0,0,0,0], [9E9, 9E9, 9E9, 9E9, 9E9, 9E9]];
	VAR robtarget OpenholeUD_437 := [[461.14, -26.7, 182.13], [0.066983, 0.703927, 0.706985, -0.013112], [0,0,0,0], [9E9, 9E9, 9E9, 9E9, 9E9, 9E9]];
	VAR robtarget OpenholeUD_438 := [[465.13, -26.7, 182.43], [0.080101, 0.702555, 0.706607, -0.026585], [0,0,0,0], [9E9, 9E9, 9E9, 9E9, 9E9, 9E9]];
	VAR robtarget OpenholeUD_439 := [[469.11, -26.7, 182.72], [0.093002, 0.700964, 0.705978, -0.039936], [0,0,0,0], [9E9, 9E9, 9E9, 9E9, 9E9, 9E9]];
	VAR robtarget OpenholeUD_440 := [[473.1, -26.7, 183.02], [0.105655, 0.699169, 0.705108, -0.053124], [0,0,0,0], [9E9, 9E9, 9E9, 9E9, 9E9, 9E9]];
	VAR robtarget OpenholeUD_441 := [[477.09, -26.7, 183.31], [0.118027, 0.697187, 0.704009, -0.066113], [0,0,0,0], [9E9, 9E9, 9E9, 9E9, 9E9, 9E9]];
	VAR robtarget OpenholeUD_442 := [[481.08, -26.7, 183.6], [0.130095, 0.695036, 0.702695, -0.078869], [0,0,0,0], [9E9, 9E9, 9E9, 9E9, 9E9, 9E9]];
	VAR robtarget OpenholeUD_443 := [[485.07, -26.7, 183.9], [0.141836, 0.692736, 0.70118, -0.091362], [0,0,0,0], [9E9, 9E9, 9E9, 9E9, 9E9, 9E9]];
	VAR robtarget OpenholeUD_444 := [[489.06, -26.7, 184.19], [0.153233, 0.690304, 0.699481, -0.103567], [0,0,0,0], [9E9, 9E9, 9E9, 9E9, 9E9, 9E9]];
	VAR robtarget OpenholeUD_445 := [[493.05, -26.7, 184.49], [0.164275, 0.68776, 0.697616, -0.115462], [0,0,0,0], [9E9, 9E9, 9E9, 9E9, 9E9, 9E9]];
	VAR robtarget OpenholeUD_446 := [[497.04, -26.7, 184.78], [0.174951, 0.685122, 0.695603, -0.127029], [0,0,0,0], [9E9, 9E9, 9E9, 9E9, 9E9, 9E9]];
	VAR robtarget OpenholeUD_447 := [[501.03, -26.7, 185.08], [0.185256, 0.682408, 0.693459, -0.138256], [0,0,0,0], [9E9, 9E9, 9E9, 9E9, 9E9, 9E9]];
	VAR robtarget OpenholeUD_448 := [[505.02, -26.7, 185.37], [0.195188, 0.679633, 0.691201, -0.149132], [0,0,0,0], [9E9, 9E9, 9E9, 9E9, 9E9, 9E9]];
	VAR robtarget OpenholeUD_449 := [[509.36, -26.7, 185.69], [0.183051, 0.683002, 0.683002, -0.183051], [0,0,0,0], [9E9, 9E9, 9E9, 9E9, 9E9, 9E9]];
	VAR robtarget OpenholeUD_450 := [[513.36, -26.7, 185.68], [0.183051, 0.683002, 0.683002, -0.183051], [0,0,0,0], [9E9, 9E9, 9E9, 9E9, 9E9, 9E9]];
	VAR robtarget OpenholeUD_451 := [[517.36, -26.7, 185.67], [0.183051, 0.683002, 0.683002, -0.183051], [0,0,0,0], [9E9, 9E9, 9E9, 9E9, 9E9, 9E9]];
	VAR robtarget OpenholeUD_452 := [[521.36, -26.7, 185.66], [0.183051, 0.683002, 0.683002, -0.183051], [0,0,0,0], [9E9, 9E9, 9E9, 9E9, 9E9, 9E9]];
	VAR robtarget OpenholeUD_453 := [[525.36, -26.7, 185.64], [0.183051, 0.683002, 0.683002, -0.183051], [0,0,0,0], [9E9, 9E9, 9E9, 9E9, 9E9, 9E9]];
	VAR robtarget OpenholeUD_454 := [[529.36, -26.7, 185.63], [0.183051, 0.683002, 0.683002, -0.183051], [0,0,0,0], [9E9, 9E9, 9E9, 9E9, 9E9, 9E9]];
	VAR robtarget OpenholeUD_455 := [[529.36, -26.7, 185.63], [0.183051, 0.683002, 0.683002, -0.183051], [0,0,0,0], [9E9, 9E9, 9E9, 9E9, 9E9, 9E9]];
	VAR robtarget OpenholeUD_456 := [[529.36, -25.5, 184.94], [0.183051, 0.683002, 0.683002, -0.183051], [0,0,0,0], [9E9, 9E9, 9E9, 9E9, 9E9, 9E9]];
	VAR robtarget OpenholeUD_457 := [[525.36, -25.5, 184.95], [0.183051, 0.683002, 0.683002, -0.183051], [0,0,0,0], [9E9, 9E9, 9E9, 9E9, 9E9, 9E9]];
	VAR robtarget OpenholeUD_458 := [[521.36, -25.5, 184.96], [0.183051, 0.683002, 0.683002, -0.183051], [0,0,0,0], [9E9, 9E9, 9E9, 9E9, 9E9, 9E9]];
	VAR robtarget OpenholeUD_459 := [[517.36, -25.5, 184.97], [0.183051, 0.683002, 0.683002, -0.183051], [0,0,0,0], [9E9, 9E9, 9E9, 9E9, 9E9, 9E9]];
	VAR robtarget OpenholeUD_460 := [[513.36, -25.5, 184.99], [0.183051, 0.683002, 0.683002, -0.183051], [0,0,0,0], [9E9, 9E9, 9E9, 9E9, 9E9, 9E9]];
	VAR robtarget OpenholeUD_461 := [[509.36, -25.5, 185], [0.183051, 0.683002, 0.683002, -0.183051], [0,0,0,0], [9E9, 9E9, 9E9, 9E9, 9E9, 9E9]];
	VAR robtarget OpenholeUD_462 := [[505.37, -25.5, 184.75], [0.192602, 0.680371, 0.69023, -0.153567], [0,0,0,0], [9E9, 9E9, 9E9, 9E9, 9E9, 9E9]];
	VAR robtarget OpenholeUD_463 := [[501.37, -25.5, 184.5], [0.182626, 0.683116, 0.692542, -0.14278], [0,0,0,0], [9E9, 9E9, 9E9, 9E9, 9E9, 9E9]];
	VAR robtarget OpenholeUD_464 := [[497.38, -25.5, 184.25], [0.172278, 0.685799, 0.694745, -0.131639], [0,0,0,0], [9E9, 9E9, 9E9, 9E9, 9E9, 9E9]];
	VAR robtarget OpenholeUD_465 := [[493.39, -25.5, 184.01], [0.16156, 0.688403, 0.696824, -0.120153], [0,0,0,0], [9E9, 9E9, 9E9, 9E9, 9E9, 9E9]];
	VAR robtarget OpenholeUD_466 := [[489.4, -25.5, 183.76], [0.150478, 0.69091, 0.698758, -0.108336], [0,0,0,0], [9E9, 9E9, 9E9, 9E9, 9E9, 9E9]];
	VAR robtarget OpenholeUD_467 := [[485.4, -25.5, 183.51], [0.139042, 0.693302, 0.700532, -0.096202], [0,0,0,0], [9E9, 9E9, 9E9, 9E9, 9E9, 9E9]];
	VAR robtarget OpenholeUD_468 := [[481.41, -25.5, 183.26], [0.127264, 0.69556, 0.702127, -0.083774], [0,0,0,0], [9E9, 9E9, 9E9, 9E9, 9E9, 9E9]];
	VAR robtarget OpenholeUD_469 := [[477.42, -25.5, 183.01], [0.115163, 0.697666, 0.703526, -0.071075], [0,0,0,0], [9E9, 9E9, 9E9, 9E9, 9E9, 9E9]];
	VAR robtarget OpenholeUD_470 := [[473.43, -25.5, 182.76], [0.102758, 0.6996, 0.704713, -0.058135], [0,0,0,0], [9E9, 9E9, 9E9, 9E9, 9E9, 9E9]];
	VAR robtarget OpenholeUD_471 := [[469.44, -25.5, 182.51], [0.090077, 0.701346, 0.705674, -0.044987], [0,0,0,0], [9E9, 9E9, 9E9, 9E9, 9E9, 9E9]];
	VAR robtarget OpenholeUD_472 := [[465.44, -25.5, 182.26], [0.077149, 0.702886, 0.706397, -0.031667], [0,0,0,0], [9E9, 9E9, 9E9, 9E9, 9E9, 9E9]];
	VAR robtarget OpenholeUD_473 := [[461.45, -25.5, 182.02], [0.064008, 0.704204, 0.706872, -0.018214], [0,0,0,0], [9E9, 9E9, 9E9, 9E9, 9E9, 9E9]];
	VAR robtarget OpenholeUD_474 := [[457.46, -25.5, 181.77], [0.050691, 0.705287, 0.707091, -0.004671], [0,0,0,0], [9E9, 9E9, 9E9, 9E9, 9E9, 9E9]];
	VAR robtarget OpenholeUD_475 := [[453.47, -25.5, 181.52], [0.03724, 0.706125, 0.707051, 0.008918], [0,0,0,0], [9E9, 9E9, 9E9, 9E9, 9E9, 9E9]];
	VAR robtarget OpenholeUD_476 := [[449.47, -25.5, 181.27], [0.023697, 0.70671, 0.706748, 0.022509], [0,0,0,0], [9E9, 9E9, 9E9, 9E9, 9E9, 9E9]];
	VAR robtarget OpenholeUD_477 := [[445.48, -25.5, 181.02], [0.010106, 0.707035, 0.706187, 0.036056], [0,0,0,0], [9E9, 9E9, 9E9, 9E9, 9E9, 9E9]];
	VAR robtarget OpenholeUD_478 := [[441.49, -25.5, 180.77], [-0.003487, 0.707098, 0.705371, 0.049514], [0,0,0,0], [9E9, 9E9, 9E9, 9E9, 9E9, 9E9]];
	VAR robtarget OpenholeUD_479 := [[437.5, -25.5, 180.52], [-0.017038, 0.706901, 0.704309, 0.062842], [0,0,0,0], [9E9, 9E9, 9E9, 9E9, 9E9, 9E9]];
	VAR robtarget OpenholeUD_480 := [[433.51, -25.5, 180.27], [-0.030502, 0.706449, 0.703011, 0.075998], [0,0,0,0], [9E9, 9E9, 9E9, 9E9, 9E9, 9E9]];
	VAR robtarget OpenholeUD_481 := [[429.51, -25.5, 180.03], [-0.043838, 0.705747, 0.701491, 0.088944], [0,0,0,0], [9E9, 9E9, 9E9, 9E9, 9E9, 9E9]];
	VAR robtarget OpenholeUD_482 := [[425.52, -25.5, 179.78], [-0.057005, 0.704805, 0.699763, 0.101647], [0,0,0,0], [9E9, 9E9, 9E9, 9E9, 9E9, 9E9]];
	VAR robtarget OpenholeUD_483 := [[421.53, -25.5, 179.53], [-0.069966, 0.703637, 0.697844, 0.114075], [0,0,0,0], [9E9, 9E9, 9E9, 9E9, 9E9, 9E9]];
	VAR robtarget OpenholeUD_484 := [[417.54, -25.5, 179.28], [-0.082688, 0.702255, 0.695753, 0.126203], [0,0,0,0], [9E9, 9E9, 9E9, 9E9, 9E9, 9E9]];
	VAR robtarget OpenholeUD_485 := [[413.54, -25.5, 179.03], [-0.095143, 0.700677, 0.693508, 0.138009], [0,0,0,0], [9E9, 9E9, 9E9, 9E9, 9E9, 9E9]];
	VAR robtarget OpenholeUD_486 := [[409.55, -25.5, 178.78], [-0.107304, 0.698918, 0.691128, 0.149474], [0,0,0,0], [9E9, 9E9, 9E9, 9E9, 9E9, 9E9]];
	VAR robtarget OpenholeUD_487 := [[405.56, -25.5, 178.53], [-0.119151, 0.696996, 0.688631, 0.160586], [0,0,0,0], [9E9, 9E9, 9E9, 9E9, 9E9, 9E9]];
	VAR robtarget OpenholeUD_488 := [[401.57, -25.5, 178.29], [-0.130667, 0.694929, 0.686035, 0.171335], [0,0,0,0], [9E9, 9E9, 9E9, 9E9, 9E9, 9E9]];
	VAR robtarget OpenholeUD_489 := [[397.57, -25.5, 178.04], [-0.141839, 0.692735, 0.683359, 0.181715], [0,0,0,0], [9E9, 9E9, 9E9, 9E9, 9E9, 9E9]];
	VAR robtarget OpenholeUD_490 := [[393.58, -25.5, 177.79], [-0.152658, 0.690431, 0.680619, 0.191724], [0,0,0,0], [9E9, 9E9, 9E9, 9E9, 9E9, 9E9]];
	VAR robtarget OpenholeUD_491 := [[389.33, -25.5, 177.52], [-0.163778, 0.687879, 0.67765, 0.201967], [0,0,0,0], [9E9, 9E9, 9E9, 9E9, 9E9, 9E9]];
	VAR robtarget OpenholeUD_492 := [[385.33, -25.5, 177.54], [-0.183051, 0.683002, 0.683002, 0.183051], [0,0,0,0], [9E9, 9E9, 9E9, 9E9, 9E9, 9E9]];
	VAR robtarget OpenholeUD_493 := [[381.33, -25.5, 177.55], [-0.183051, 0.683002, 0.683002, 0.183051], [0,0,0,0], [9E9, 9E9, 9E9, 9E9, 9E9, 9E9]];
	VAR robtarget OpenholeUD_494 := [[377.33, -25.5, 177.56], [-0.183051, 0.683002, 0.683002, 0.183051], [0,0,0,0], [9E9, 9E9, 9E9, 9E9, 9E9, 9E9]];
	VAR robtarget OpenholeUD_495 := [[373.33, -25.5, 177.57], [-0.183051, 0.683002, 0.683002, 0.183051], [0,0,0,0], [9E9, 9E9, 9E9, 9E9, 9E9, 9E9]];
	VAR robtarget OpenholeUD_496 := [[369.33, -25.5, 177.59], [-0.183051, 0.683002, 0.683002, 0.183051], [0,0,0,0], [9E9, 9E9, 9E9, 9E9, 9E9, 9E9]];
	VAR robtarget OpenholeUD_497 := [[369.33, -25.5, 177.59], [-0.183051, 0.683002, 0.683002, 0.183051], [0,0,0,0], [9E9, 9E9, 9E9, 9E9, 9E9, 9E9]];
	VAR robtarget OpenholeUD_498 := [[369.34, -24.3, 178.28], [-0.183051, 0.683002, 0.683002, 0.183051], [0,0,0,0], [9E9, 9E9, 9E9, 9E9, 9E9, 9E9]];
	VAR robtarget OpenholeUD_499 := [[373.34, -24.3, 178.27], [-0.183051, 0.683002, 0.683002, 0.183051], [0,0,0,0], [9E9, 9E9, 9E9, 9E9, 9E9, 9E9]];
	VAR robtarget OpenholeUD_500 := [[377.34, -24.3, 178.25], [-0.183051, 0.683002, 0.683002, 0.183051], [0,0,0,0], [9E9, 9E9, 9E9, 9E9, 9E9, 9E9]];
	VAR robtarget OpenholeUD_501 := [[381.34, -24.3, 178.24], [-0.183051, 0.683002, 0.683002, 0.183051], [0,0,0,0], [9E9, 9E9, 9E9, 9E9, 9E9, 9E9]];
	VAR robtarget OpenholeUD_502 := [[389.34, -24.3, 178.22], [-0.167207, 0.687053, 0.67865, 0.198582], [0,0,0,0], [9E9, 9E9, 9E9, 9E9, 9E9, 9E9]];
	VAR robtarget OpenholeUD_503 := [[393.33, -24.3, 178.42], [-0.156831, 0.689495, 0.68141, 0.188892], [0,0,0,0], [9E9, 9E9, 9E9, 9E9, 9E9, 9E9]];
	VAR robtarget OpenholeUD_504 := [[397.33, -24.3, 178.62], [-0.146094, 0.69185, 0.684119, 0.178832], [0,0,0,0], [9E9, 9E9, 9E9, 9E9, 9E9, 9E9]];
	VAR robtarget OpenholeUD_505 := [[401.32, -24.3, 178.82], [-0.135002, 0.6941, 0.686761, 0.168402], [0,0,0,0], [9E9, 9E9, 9E9, 9E9, 9E9, 9E9]];
	VAR robtarget OpenholeUD_506 := [[405.32, -24.3, 179.03], [-0.123562, 0.696227, 0.689319, 0.157603], [0,0,0,0], [9E9, 9E9, 9E9, 9E9, 9E9, 9E9]];
	VAR robtarget OpenholeUD_507 := [[409.31, -24.3, 179.23], [-0.111786, 0.698215, 0.691776, 0.146444], [0,0,0,0], [9E9, 9E9, 9E9, 9E9, 9E9, 9E9]];
	VAR robtarget OpenholeUD_508 := [[413.31, -24.3, 179.43], [-0.099692, 0.700044, 0.694113, 0.134932], [0,0,0,0], [9E9, 9E9, 9E9, 9E9, 9E9, 9E9]];
	VAR robtarget OpenholeUD_509 := [[417.3, -24.3, 179.64], [-0.087298, 0.701697, 0.696312, 0.123084], [0,0,0,0], [9E9, 9E9, 9E9, 9E9, 9E9, 9E9]];
	VAR robtarget OpenholeUD_510 := [[421.3, -24.3, 179.84], [-0.074629, 0.703158, 0.698354, 0.110915], [0,0,0,0], [9E9, 9E9, 9E9, 9E9, 9E9, 9E9]];
	VAR robtarget OpenholeUD_511 := [[425.29, -24.3, 180.04], [-0.061714, 0.704409, 0.70022, 0.09845], [0,0,0,0], [9E9, 9E9, 9E9, 9E9, 9E9, 9E9]];
	VAR robtarget OpenholeUD_512 := [[429.28, -24.3, 180.24], [-0.048585, 0.705436, 0.701893, 0.085714], [0,0,0,0], [9E9, 9E9, 9E9, 9E9, 9E9, 9E9]];
	VAR robtarget OpenholeUD_513 := [[433.28, -24.3, 180.45], [-0.035279, 0.706226, 0.703356, 0.072738], [0,0,0,0], [9E9, 9E9, 9E9, 9E9, 9E9, 9E9]];
	VAR robtarget OpenholeUD_514 := [[437.27, -24.3, 180.65], [-0.021835, 0.70677, 0.704594, 0.059556], [0,0,0,0], [9E9, 9E9, 9E9, 9E9, 9E9, 9E9]];
	VAR robtarget OpenholeUD_515 := [[441.27, -24.3, 180.85], [-0.008295, 0.707058, 0.705595, 0.046207], [0,0,0,0], [9E9, 9E9, 9E9, 9E9, 9E9, 9E9]];
	VAR robtarget OpenholeUD_516 := [[446.05, -24.3, 181.09], [0.007958, 0.707062, 0.706466, 0.030086], [0,0,0,0], [9E9, 9E9, 9E9, 9E9, 9E9, 9E9]];
	VAR robtarget OpenholeUD_517 := [[446.05, -24.3, 181.09], [0.007958, 0.707062, 0.706466, 0.030086], [0,0,0,0], [9E9, 9E9, 9E9, 9E9, 9E9, 9E9]];
	VAR robtarget OpenholeUD_518 := [[444.56, -23.1, 181.07], [-0.001167, 0.707106, 0.706425, 0.031047], [0,0,0,0], [9E9, 9E9, 9E9, 9E9, 9E9, 9E9]];
	VAR robtarget OpenholeUD_519 := [[440.56, -23.1, 180.92], [-0.014751, 0.706953, 0.705704, 0.044525], [0,0,0,0], [9E9, 9E9, 9E9, 9E9, 9E9, 9E9]];
	VAR robtarget OpenholeUD_520 := [[436.57, -23.1, 180.76], [-0.028267, 0.706542, 0.704734, 0.057876], [0,0,0,0], [9E9, 9E9, 9E9, 9E9, 9E9, 9E9]];
	VAR robtarget OpenholeUD_521 := [[432.57, -23.1, 180.6], [-0.041673, 0.705878, 0.703527, 0.071059], [0,0,0,0], [9E9, 9E9, 9E9, 9E9, 9E9, 9E9]];
	VAR robtarget OpenholeUD_522 := [[428.57, -23.1, 180.45], [-0.054926, 0.70497, 0.702095, 0.084037], [0,0,0,0], [9E9, 9E9, 9E9, 9E9, 9E9, 9E9]];
	VAR robtarget OpenholeUD_523 := [[424.58, -23.1, 180.29], [-0.067988, 0.703831, 0.700453, 0.096775], [0,0,0,0], [9E9, 9E9, 9E9, 9E9, 9E9, 9E9]];
	VAR robtarget OpenholeUD_524 := [[420.58, -23.1, 180.13], [-0.080825, 0.702472, 0.698617, 0.109242], [0,0,0,0], [9E9, 9E9, 9E9, 9E9, 9E9, 9E9]];
	VAR robtarget OpenholeUD_525 := [[416.58, -23.1, 179.98], [-0.093404, 0.700911, 0.696605, 0.121412], [0,0,0,0], [9E9, 9E9, 9E9, 9E9, 9E9, 9E9]];
	VAR robtarget OpenholeUD_526 := [[412.59, -23.1, 179.82], [-0.105699, 0.699162, 0.694436, 0.133264], [0,0,0,0], [9E9, 9E9, 9E9, 9E9, 9E9, 9E9]];
	VAR robtarget OpenholeUD_527 := [[408.59, -23.1, 179.66], [-0.117687, 0.697244, 0.692127, 0.144778], [0,0,0,0], [9E9, 9E9, 9E9, 9E9, 9E9, 9E9]];
	VAR robtarget OpenholeUD_528 := [[404.59, -23.1, 179.51], [-0.129348, 0.695176, 0.689697, 0.155941], [0,0,0,0], [9E9, 9E9, 9E9, 9E9, 9E9, 9E9]];
	VAR robtarget OpenholeUD_529 := [[400.59, -23.1, 179.35], [-0.140668, 0.692974, 0.687165, 0.166744], [0,0,0,0], [9E9, 9E9, 9E9, 9E9, 9E9, 9E9]];
	VAR robtarget OpenholeUD_530 := [[396.6, -23.1, 179.19], [-0.151636, 0.690657, 0.684549, 0.17718], [0,0,0,0], [9E9, 9E9, 9E9, 9E9, 9E9, 9E9]];
	VAR robtarget OpenholeUD_531 := [[389.34, -23.1, 178.91], [-0.170635, 0.68621, 0.679633, 0.195189], [0,0,0,0], [9E9, 9E9, 9E9, 9E9, 9E9, 9E9]];
	VAR robtarget OpenholeUD_532 := [[385.34, -23.1, 178.92], [-0.183051, 0.683002, 0.683002, 0.183051], [0,0,0,0], [9E9, 9E9, 9E9, 9E9, 9E9, 9E9]];
	VAR robtarget OpenholeUD_533 := [[381.34, -23.1, 178.93], [-0.183051, 0.683002, 0.683002, 0.183051], [0,0,0,0], [9E9, 9E9, 9E9, 9E9, 9E9, 9E9]];
	VAR robtarget OpenholeUD_534 := [[377.34, -23.1, 178.95], [-0.183051, 0.683002, 0.683002, 0.183051], [0,0,0,0], [9E9, 9E9, 9E9, 9E9, 9E9, 9E9]];
	VAR robtarget OpenholeUD_535 := [[373.34, -23.1, 178.96], [-0.183051, 0.683002, 0.683002, 0.183051], [0,0,0,0], [9E9, 9E9, 9E9, 9E9, 9E9, 9E9]];
	VAR robtarget OpenholeUD_536 := [[369.34, -23.1, 178.97], [-0.183051, 0.683002, 0.683002, 0.183051], [0,0,0,0], [9E9, 9E9, 9E9, 9E9, 9E9, 9E9]];
	VAR robtarget OpenholeUD_537 := [[369.34, -23.1, 178.97], [-0.183051, 0.683002, 0.683002, 0.183051], [0,0,0,0], [9E9, 9E9, 9E9, 9E9, 9E9, 9E9]];
	VAR robtarget OpenholeUD_538 := [[369.34, -21.9, 179.66], [-0.183051, 0.683002, 0.683002, 0.183051], [0,0,0,0], [9E9, 9E9, 9E9, 9E9, 9E9, 9E9]];
	VAR robtarget OpenholeUD_539 := [[373.34, -21.9, 179.65], [-0.183051, 0.683002, 0.683002, 0.183051], [0,0,0,0], [9E9, 9E9, 9E9, 9E9, 9E9, 9E9]];
	VAR robtarget OpenholeUD_540 := [[377.34, -21.9, 179.64], [-0.183051, 0.683002, 0.683002, 0.183051], [0,0,0,0], [9E9, 9E9, 9E9, 9E9, 9E9, 9E9]];
	VAR robtarget OpenholeUD_541 := [[381.34, -21.9, 179.63], [-0.183051, 0.683002, 0.683002, 0.183051], [0,0,0,0], [9E9, 9E9, 9E9, 9E9, 9E9, 9E9]];
	VAR robtarget OpenholeUD_542 := [[385.34, -21.9, 179.61], [-0.183051, 0.683002, 0.683002, 0.183051], [0,0,0,0], [9E9, 9E9, 9E9, 9E9, 9E9, 9E9]];
	VAR robtarget OpenholeUD_543 := [[389.34, -21.9, 179.6], [-0.174061, 0.685349, 0.680601, 0.191788], [0,0,0,0], [9E9, 9E9, 9E9, 9E9, 9E9, 9E9]];
	VAR robtarget OpenholeUD_544 := [[393.34, -21.9, 179.71], [-0.163813, 0.68787, 0.683296, 0.18195], [0,0,0,0], [9E9, 9E9, 9E9, 9E9, 9E9, 9E9]];
	VAR robtarget OpenholeUD_545 := [[397.34, -21.9, 179.82], [-0.153202, 0.690311, 0.685933, 0.171743], [0,0,0,0], [9E9, 9E9, 9E9, 9E9, 9E9, 9E9]];
	VAR robtarget OpenholeUD_546 := [[401.34, -21.9, 179.93], [-0.142229, 0.692655, 0.688495, 0.161168], [0,0,0,0], [9E9, 9E9, 9E9, 9E9, 9E9, 9E9]];
	VAR robtarget OpenholeUD_547 := [[405.33, -21.9, 180.04], [-0.130904, 0.694884, 0.690964, 0.150229], [0,0,0,0], [9E9, 9E9, 9E9, 9E9, 9E9, 9E9]];
	VAR robtarget OpenholeUD_548 := [[409.33, -21.9, 180.15], [-0.119237, 0.696981, 0.693324, 0.138932], [0,0,0,0], [9E9, 9E9, 9E9, 9E9, 9E9, 9E9]];
	VAR robtarget OpenholeUD_549 := [[413.33, -21.9, 180.27], [-0.107243, 0.698927, 0.695555, 0.127291], [0,0,0,0], [9E9, 9E9, 9E9, 9E9, 9E9, 9E9]];
	VAR robtarget OpenholeUD_550 := [[417.33, -21.9, 180.38], [-0.094941, 0.700704, 0.69764, 0.115319], [0,0,0,0], [9E9, 9E9, 9E9, 9E9, 9E9, 9E9]];
	VAR robtarget OpenholeUD_551 := [[421.33, -21.9, 180.49], [-0.082354, 0.702295, 0.69956, 0.103036], [0,0,0,0], [9E9, 9E9, 9E9, 9E9, 9E9, 9E9]];
	VAR robtarget OpenholeUD_552 := [[425.33, -21.9, 180.6], [-0.069511, 0.703682, 0.701296, 0.090465], [0,0,0,0], [9E9, 9E9, 9E9, 9E9, 9E9, 9E9]];
	VAR robtarget OpenholeUD_553 := [[429.33, -21.9, 180.71], [-0.056441, 0.704851, 0.702832, 0.077635], [0,0,0,0], [9E9, 9E9, 9E9, 9E9, 9E9, 9E9]];
	VAR robtarget OpenholeUD_554 := [[433.32, -21.9, 180.82], [-0.043182, 0.705787, 0.704152, 0.064577], [0,0,0,0], [9E9, 9E9, 9E9, 9E9, 9E9, 9E9]];
	VAR robtarget OpenholeUD_555 := [[437.32, -21.9, 180.93], [-0.029771, 0.70648, 0.705241, 0.051327], [0,0,0,0], [9E9, 9E9, 9E9, 9E9, 9E9, 9E9]];
	VAR robtarget OpenholeUD_556 := [[443.69, -21.9, 181.1], [-0.008212, 0.707059, 0.706473, 0.029933], [0,0,0,0], [9E9, 9E9, 9E9, 9E9, 9E9, 9E9]];
	VAR robtarget OpenholeUD_557 := [[443.69, -21.9, 181.1], [-0.008212, 0.707059, 0.706473, 0.029933], [0,0,0,0], [9E9, 9E9, 9E9, 9E9, 9E9, 9E9]];
	VAR robtarget OpenholeUD_558 := [[443.16, -20.7, 181.16], [-0.014077, 0.706967, 0.706566, 0.027646], [0,0,0,0], [9E9, 9E9, 9E9, 9E9, 9E9, 9E9]];
	VAR robtarget OpenholeUD_559 := [[439.16, -20.7, 181.1], [-0.027624, 0.706567, 0.70591, 0.041126], [0,0,0,0], [9E9, 9E9, 9E9, 9E9, 9E9, 9E9]];
	VAR robtarget OpenholeUD_560 := [[435.16, -20.7, 181.03], [-0.041073, 0.705913, 0.705005, 0.054479], [0,0,0,0], [9E9, 9E9, 9E9, 9E9, 9E9, 9E9]];
	VAR robtarget OpenholeUD_561 := [[431.16, -20.7, 180.97], [-0.054383, 0.705012, 0.703862, 0.067663], [0,0,0,0], [9E9, 9E9, 9E9, 9E9, 9E9, 9E9]];
	VAR robtarget OpenholeUD_562 := [[427.16, -20.7, 180.9], [-0.067513, 0.703876, 0.702493, 0.080643], [0,0,0,0], [9E9, 9E9, 9E9, 9E9, 9E9, 9E9]];
	VAR robtarget OpenholeUD_563 := [[423.16, -20.7, 180.84], [-0.080427, 0.702518, 0.700914, 0.093382], [0,0,0,0], [9E9, 9E9, 9E9, 9E9, 9E9, 9E9]];
	VAR robtarget OpenholeUD_564 := [[419.16, -20.7, 180.78], [-0.093092, 0.700952, 0.699139, 0.105851], [0,0,0,0], [9E9, 9E9, 9E9, 9E9, 9E9, 9E9]];
	VAR robtarget OpenholeUD_565 := [[415.16, -20.7, 180.71], [-0.10548, 0.699195, 0.697187, 0.118025], [0,0,0,0], [9E9, 9E9, 9E9, 9E9, 9E9, 9E9]];
	VAR robtarget OpenholeUD_566 := [[411.16, -20.7, 180.65], [-0.117566, 0.697265, 0.695076, 0.12988], [0,0,0,0], [9E9, 9E9, 9E9, 9E9, 9E9, 9E9]];
	VAR robtarget OpenholeUD_567 := [[407.17, -20.7, 180.58], [-0.129328, 0.695179, 0.692825, 0.141399], [0,0,0,0], [9E9, 9E9, 9E9, 9E9, 9E9, 9E9]];
	VAR robtarget OpenholeUD_568 := [[403.17, -20.7, 180.52], [-0.140752, 0.692957, 0.690451, 0.152569], [0,0,0,0], [9E9, 9E9, 9E9, 9E9, 9E9, 9E9]];
	VAR robtarget OpenholeUD_569 := [[399.17, -20.7, 180.45], [-0.151824, 0.690615, 0.687973, 0.163381], [0,0,0,0], [9E9, 9E9, 9E9, 9E9, 9E9, 9E9]];
	VAR robtarget OpenholeUD_570 := [[395.17, -20.7, 180.39], [-0.162537, 0.688173, 0.685408, 0.173827], [0,0,0,0], [9E9, 9E9, 9E9, 9E9, 9E9, 9E9]];
	VAR robtarget OpenholeUD_571 := [[389.34, -20.7, 180.29], [-0.177485, 0.68447, 0.681551, 0.188381], [0,0,0,0], [9E9, 9E9, 9E9, 9E9, 9E9, 9E9]];
	VAR robtarget OpenholeUD_572 := [[385.34, -20.7, 180.31], [-0.183051, 0.683002, 0.683002, 0.183051], [0,0,0,0], [9E9, 9E9, 9E9, 9E9, 9E9, 9E9]];
	VAR robtarget OpenholeUD_573 := [[381.34, -20.7, 180.32], [-0.183051, 0.683002, 0.683002, 0.183051], [0,0,0,0], [9E9, 9E9, 9E9, 9E9, 9E9, 9E9]];
	VAR robtarget OpenholeUD_574 := [[377.34, -20.7, 180.33], [-0.183051, 0.683002, 0.683002, 0.183051], [0,0,0,0], [9E9, 9E9, 9E9, 9E9, 9E9, 9E9]];
	VAR robtarget OpenholeUD_575 := [[373.34, -20.7, 180.35], [-0.183051, 0.683002, 0.683002, 0.183051], [0,0,0,0], [9E9, 9E9, 9E9, 9E9, 9E9, 9E9]];
	VAR robtarget OpenholeUD_576 := [[369.34, -20.7, 180.36], [-0.183051, 0.683002, 0.683002, 0.183051], [0,0,0,0], [9E9, 9E9, 9E9, 9E9, 9E9, 9E9]];
	VAR robtarget OpenholeUD_577 := [[369.34, -20.7, 180.36], [-0.183051, 0.683002, 0.683002, 0.183051], [0,0,0,0], [9E9, 9E9, 9E9, 9E9, 9E9, 9E9]];
	VAR robtarget OpenholeUD_578 := [[369.34, -19.5, 181.05], [-0.183051, 0.683002, 0.683002, 0.183051], [0,0,0,0], [9E9, 9E9, 9E9, 9E9, 9E9, 9E9]];
	VAR robtarget OpenholeUD_579 := [[373.34, -19.5, 181.04], [-0.183051, 0.683002, 0.683002, 0.183051], [0,0,0,0], [9E9, 9E9, 9E9, 9E9, 9E9, 9E9]];
	VAR robtarget OpenholeUD_580 := [[377.34, -19.5, 181.03], [-0.183051, 0.683002, 0.683002, 0.183051], [0,0,0,0], [9E9, 9E9, 9E9, 9E9, 9E9, 9E9]];
	VAR robtarget OpenholeUD_581 := [[381.34, -19.5, 181.01], [-0.183051, 0.683002, 0.683002, 0.183051], [0,0,0,0], [9E9, 9E9, 9E9, 9E9, 9E9, 9E9]];
	VAR robtarget OpenholeUD_582 := [[385.34, -19.5, 181], [-0.183051, 0.683002, 0.683002, 0.183051], [0,0,0,0], [9E9, 9E9, 9E9, 9E9, 9E9, 9E9]];
	VAR robtarget OpenholeUD_583 := [[389.34, -19.5, 180.99], [-0.180905, 0.683574, 0.682486, 0.184969], [0,0,0,0], [9E9, 9E9, 9E9, 9E9, 9E9, 9E9]];
	VAR robtarget OpenholeUD_584 := [[393.34, -19.5, 181.01], [-0.170792, 0.68617, 0.685113, 0.174987], [0,0,0,0], [9E9, 9E9, 9E9, 9E9, 9E9, 9E9]];
	VAR robtarget OpenholeUD_585 := [[397.34, -19.5, 181.02], [-0.160312, 0.688694, 0.687673, 0.164638], [0,0,0,0], [9E9, 9E9, 9E9, 9E9, 9E9, 9E9]];
	VAR robtarget OpenholeUD_586 := [[401.34, -19.5, 181.04], [-0.149468, 0.691129, 0.69015, 0.153925], [0,0,0,0], [9E9, 9E9, 9E9, 9E9, 9E9, 9E9]];
	VAR robtarget OpenholeUD_587 := [[405.34, -19.5, 181.06], [-0.138266, 0.693457, 0.692527, 0.142851], [0,0,0,0], [9E9, 9E9, 9E9, 9E9, 9E9, 9E9]];
	VAR robtarget OpenholeUD_588 := [[409.34, -19.5, 181.08], [-0.126715, 0.69566, 0.694786, 0.131426], [0,0,0,0], [9E9, 9E9, 9E9, 9E9, 9E9, 9E9]];
	VAR robtarget OpenholeUD_589 := [[413.34, -19.5, 181.1], [-0.114831, 0.69772, 0.696908, 0.119661], [0,0,0,0], [9E9, 9E9, 9E9, 9E9, 9E9, 9E9]];
	VAR robtarget OpenholeUD_590 := [[417.34, -19.5, 181.12], [-0.10263, 0.699619, 0.698876, 0.107574], [0,0,0,0], [9E9, 9E9, 9E9, 9E9, 9E9, 9E9]];
	VAR robtarget OpenholeUD_591 := [[421.34, -19.5, 181.13], [-0.090135, 0.701339, 0.700671, 0.095185], [0,0,0,0], [9E9, 9E9, 9E9, 9E9, 9E9, 9E9]];
	VAR robtarget OpenholeUD_592 := [[425.34, -19.5, 181.15], [-0.077372, 0.702861, 0.702275, 0.082519], [0,0,0,0], [9E9, 9E9, 9E9, 9E9, 9E9, 9E9]];
	VAR robtarget OpenholeUD_593 := [[429.34, -19.5, 181.17], [-0.064372, 0.704171, 0.703673, 0.069604], [0,0,0,0], [9E9, 9E9, 9E9, 9E9, 9E9, 9E9]];
	VAR robtarget OpenholeUD_594 := [[433.34, -19.5, 181.19], [-0.051169, 0.705253, 0.704848, 0.056473], [0,0,0,0], [9E9, 9E9, 9E9, 9E9, 9E9, 9E9]];
	VAR robtarget OpenholeUD_595 := [[437.34, -19.5, 181.21], [-0.037801, 0.706096, 0.705788, 0.043164], [0,0,0,0], [9E9, 9E9, 9E9, 9E9, 9E9, 9E9]];
	VAR robtarget OpenholeUD_596 := [[442.9, -19.5, 181.23], [-0.019054, 0.70685, 0.706683, 0.024472], [0,0,0,0], [9E9, 9E9, 9E9, 9E9, 9E9, 9E9]];
	VAR robtarget OpenholeUD_597 := [[442.9, -19.5, 181.23], [-0.019054, 0.70685, 0.706683, 0.024472], [0,0,0,0], [9E9, 9E9, 9E9, 9E9, 9E9, 9E9]];
	VAR robtarget OpenholeUD_598 := [[442.86, -18.3, 181.31], [-0.023254, 0.706724, 0.706809, 0.020524], [0,0,0,0], [9E9, 9E9, 9E9, 9E9, 9E9, 9E9]];
	VAR robtarget OpenholeUD_599 := [[438.86, -18.3, 181.33], [-0.036766, 0.70615, 0.706287, 0.034031], [0,0,0,0], [9E9, 9E9, 9E9, 9E9, 9E9, 9E9]];
	VAR robtarget OpenholeUD_600 := [[434.86, -18.3, 181.36], [-0.050163, 0.705325, 0.705515, 0.047421], [0,0,0,0], [9E9, 9E9, 9E9, 9E9, 9E9, 9E9]];
	VAR robtarget OpenholeUD_601 := [[430.86, -18.3, 181.39], [-0.063404, 0.704258, 0.704501, 0.060654], [0,0,0,0], [9E9, 9E9, 9E9, 9E9, 9E9, 9E9]];
	VAR robtarget OpenholeUD_602 := [[426.86, -18.3, 181.42], [-0.076449, 0.702962, 0.703256, 0.073691], [0,0,0,0], [9E9, 9E9, 9E9, 9E9, 9E9, 9E9]];
	VAR robtarget OpenholeUD_603 := [[422.86, -18.3, 181.45], [-0.089263, 0.70145, 0.701796, 0.086497], [0,0,0,0], [9E9, 9E9, 9E9, 9E9, 9E9, 9E9]];
	VAR robtarget OpenholeUD_604 := [[418.86, -18.3, 181.47], [-0.101816, 0.699738, 0.700136, 0.099042], [0,0,0,0], [9E9, 9E9, 9E9, 9E9, 9E9, 9E9]];
	VAR robtarget OpenholeUD_605 := [[414.86, -18.3, 181.5], [-0.114079, 0.697844, 0.698293, 0.111299], [0,0,0,0], [9E9, 9E9, 9E9, 9E9, 9E9, 9E9]];
	VAR robtarget OpenholeUD_606 := [[410.86, -18.3, 181.53], [-0.126029, 0.695785, 0.696284, 0.123244], [0,0,0,0], [9E9, 9E9, 9E9, 9E9, 9E9, 9E9]];
	VAR robtarget OpenholeUD_607 := [[406.86, -18.3, 181.56], [-0.137647, 0.69358, 0.694127, 0.13486], [0,0,0,0], [9E9, 9E9, 9E9, 9E9, 9E9, 9E9]];
	VAR robtarget OpenholeUD_608 := [[402.86, -18.3, 181.59], [-0.148919, 0.691248, 0.691842, 0.146131], [0,0,0,0], [9E9, 9E9, 9E9, 9E9, 9E9, 9E9]];
	VAR robtarget OpenholeUD_609 := [[398.86, -18.3, 181.61], [-0.159834, 0.688806, 0.689446, 0.157048], [0,0,0,0], [9E9, 9E9, 9E9, 9E9, 9E9, 9E9]];
	VAR robtarget OpenholeUD_610 := [[394.86, -18.3, 181.64], [-0.170384, 0.686272, 0.686956, 0.167603], [0,0,0,0], [9E9, 9E9, 9E9, 9E9, 9E9, 9E9]];
	VAR robtarget OpenholeUD_611 := [[389.35, -18.3, 181.68], [-0.184322, 0.682661, 0.683403, 0.181551], [0,0,0,0], [9E9, 9E9, 9E9, 9E9, 9E9, 9E9]];
	VAR robtarget OpenholeUD_612 := [[385.35, -18.3, 181.69], [-0.183051, 0.683002, 0.683002, 0.183051], [0,0,0,0], [9E9, 9E9, 9E9, 9E9, 9E9, 9E9]];
	VAR robtarget OpenholeUD_613 := [[381.35, -18.3, 181.71], [-0.183051, 0.683002, 0.683002, 0.183051], [0,0,0,0], [9E9, 9E9, 9E9, 9E9, 9E9, 9E9]];
	VAR robtarget OpenholeUD_614 := [[377.35, -18.3, 181.72], [-0.183051, 0.683002, 0.683002, 0.183051], [0,0,0,0], [9E9, 9E9, 9E9, 9E9, 9E9, 9E9]];
	VAR robtarget OpenholeUD_615 := [[373.35, -18.3, 181.73], [-0.183051, 0.683002, 0.683002, 0.183051], [0,0,0,0], [9E9, 9E9, 9E9, 9E9, 9E9, 9E9]];
	VAR robtarget OpenholeUD_616 := [[369.35, -18.3, 181.74], [-0.183051, 0.683002, 0.683002, 0.183051], [0,0,0,0], [9E9, 9E9, 9E9, 9E9, 9E9, 9E9]];
	VAR robtarget OpenholeUD_617 := [[369.35, -18.3, 181.74], [-0.183051, 0.683002, 0.683002, 0.183051], [0,0,0,0], [9E9, 9E9, 9E9, 9E9, 9E9, 9E9]];
	VAR robtarget OpenholeUD_618 := [[369.35, -17.1, 182.44], [-0.183051, 0.683002, 0.683002, 0.183051], [0,0,0,0], [9E9, 9E9, 9E9, 9E9, 9E9, 9E9]];
	VAR robtarget OpenholeUD_619 := [[373.35, -17.1, 182.42], [-0.183051, 0.683002, 0.683002, 0.183051], [0,0,0,0], [9E9, 9E9, 9E9, 9E9, 9E9, 9E9]];
	VAR robtarget OpenholeUD_620 := [[377.35, -17.1, 182.41], [-0.183051, 0.683002, 0.683002, 0.183051], [0,0,0,0], [9E9, 9E9, 9E9, 9E9, 9E9, 9E9]];
	VAR robtarget OpenholeUD_621 := [[381.35, -17.1, 182.4], [-0.183051, 0.683002, 0.683002, 0.183051], [0,0,0,0], [9E9, 9E9, 9E9, 9E9, 9E9, 9E9]];
	VAR robtarget OpenholeUD_622 := [[389.35, -17.1, 182.37], [-0.187733, 0.68173, 0.684303, 0.178129], [0,0,0,0], [9E9, 9E9, 9E9, 9E9, 9E9, 9E9]];
	VAR robtarget OpenholeUD_623 := [[393.35, -17.1, 182.3], [-0.177761, 0.684398, 0.686857, 0.168009], [0,0,0,0], [9E9, 9E9, 9E9, 9E9, 9E9, 9E9]];
	VAR robtarget OpenholeUD_624 := [[397.35, -17.1, 182.23], [-0.16742, 0.687001, 0.689337, 0.157525], [0,0,0,0], [9E9, 9E9, 9E9, 9E9, 9E9, 9E9]];
	VAR robtarget OpenholeUD_625 := [[401.35, -17.1, 182.15], [-0.15671, 0.689523, 0.691726, 0.14668], [0,0,0,0], [9E9, 9E9, 9E9, 9E9, 9E9, 9E9]];
	VAR robtarget OpenholeUD_626 := [[405.35, -17.1, 182.08], [-0.145638, 0.691946, 0.694007, 0.135479], [0,0,0,0], [9E9, 9E9, 9E9, 9E9, 9E9, 9E9]];
	VAR robtarget OpenholeUD_627 := [[409.35, -17.1, 182], [-0.134213, 0.694253, 0.696161, 0.123932], [0,0,0,0], [9E9, 9E9, 9E9, 9E9, 9E9, 9E9]];
	VAR robtarget OpenholeUD_628 := [[413.35, -17.1, 181.93], [-0.122446, 0.696424, 0.698172, 0.112053], [0,0,0,0], [9E9, 9E9, 9E9, 9E9, 9E9, 9E9]];
	VAR robtarget OpenholeUD_629 := [[417.34, -17.1, 181.85], [-0.110355, 0.698442, 0.70002, 0.09986], [0,0,0,0], [9E9, 9E9, 9E9, 9E9, 9E9, 9E9]];
	VAR robtarget OpenholeUD_630 := [[421.34, -17.1, 181.78], [-0.097961, 0.700288, 0.701688, 0.087374], [0,0,0,0], [9E9, 9E9, 9E9, 9E9, 9E9, 9E9]];
	VAR robtarget OpenholeUD_631 := [[425.34, -17.1, 181.71], [-0.085289, 0.701944, 0.703158, 0.07462], [0,0,0,0], [9E9, 9E9, 9E9, 9E9, 9E9, 9E9]];
	VAR robtarget OpenholeUD_632 := [[429.34, -17.1, 181.63], [-0.072367, 0.703394, 0.704416, 0.06163], [0,0,0,0], [9E9, 9E9, 9E9, 9E9, 9E9, 9E9]];
	VAR robtarget OpenholeUD_633 := [[433.34, -17.1, 181.56], [-0.059231, 0.704622, 0.705446, 0.048437], [0,0,0,0], [9E9, 9E9, 9E9, 9E9, 9E9, 9E9]];
	VAR robtarget OpenholeUD_634 := [[437.34, -17.1, 181.48], [-0.045916, 0.705614, 0.706236, 0.035078], [0,0,0,0], [9E9, 9E9, 9E9, 9E9, 9E9, 9E9]];
	VAR robtarget OpenholeUD_635 := [[443.05, -17.1, 181.38], [-0.026691, 0.706603, 0.70693, 0.015815], [0,0,0,0], [9E9, 9E9, 9E9, 9E9, 9E9, 9E9]];
	VAR robtarget OpenholeUD_636 := [[443.05, -17.1, 181.38], [-0.026691, 0.706603, 0.70693, 0.015815], [0,0,0,0], [9E9, 9E9, 9E9, 9E9, 9E9, 9E9]];
	VAR robtarget OpenholeUD_637 := [[443.48, -15.9, 181.44], [-0.029294, 0.7065, 0.707032, 0.010269], [0,0,0,0], [9E9, 9E9, 9E9, 9E9, 9E9, 9E9]];
	VAR robtarget OpenholeUD_638 := [[439.48, -15.9, 181.56], [-0.042786, 0.705811, 0.706706, 0.023812], [0,0,0,0], [9E9, 9E9, 9E9, 9E9, 9E9, 9E9]];
	VAR robtarget OpenholeUD_639 := [[435.48, -15.9, 181.68], [-0.056154, 0.704874, 0.706124, 0.037261], [0,0,0,0], [9E9, 9E9, 9E9, 9E9, 9E9, 9E9]];
	VAR robtarget OpenholeUD_640 := [[431.49, -15.9, 181.8], [-0.069358, 0.703697, 0.705296, 0.050572], [0,0,0,0], [9E9, 9E9, 9E9, 9E9, 9E9, 9E9]];
	VAR robtarget OpenholeUD_641 := [[427.49, -15.9, 181.92], [-0.08236, 0.702294, 0.704231, 0.063707], [0,0,0,0], [9E9, 9E9, 9E9, 9E9, 9E9, 9E9]];
	VAR robtarget OpenholeUD_642 := [[423.49, -15.9, 182.04], [-0.095125, 0.700679, 0.702942, 0.076628], [0,0,0,0], [9E9, 9E9, 9E9, 9E9, 9E9, 9E9]];
	VAR robtarget OpenholeUD_643 := [[419.49, -15.9, 182.16], [-0.107622, 0.698869, 0.701445, 0.089304], [0,0,0,0], [9E9, 9E9, 9E9, 9E9, 9E9, 9E9]];
	VAR robtarget OpenholeUD_644 := [[415.49, -15.9, 182.28], [-0.119823, 0.696881, 0.699754, 0.101706], [0,0,0,0], [9E9, 9E9, 9E9, 9E9, 9E9, 9E9]];
	VAR robtarget OpenholeUD_645 := [[411.49, -15.9, 182.4], [-0.131706, 0.694733, 0.697888, 0.113809], [0,0,0,0], [9E9, 9E9, 9E9, 9E9, 9E9, 9E9]];
	VAR robtarget OpenholeUD_646 := [[407.5, -15.9, 182.52], [-0.143254, 0.692444, 0.695864, 0.125592], [0,0,0,0], [9E9, 9E9, 9E9, 9E9, 9E9, 9E9]];
	VAR robtarget OpenholeUD_647 := [[403.5, -15.9, 182.64], [-0.154451, 0.690033, 0.6937, 0.13704], [0,0,0,0], [9E9, 9E9, 9E9, 9E9, 9E9, 9E9]];
	VAR robtarget OpenholeUD_648 := [[399.5, -15.9, 182.76], [-0.165287, 0.687517, 0.691415, 0.148139], [0,0,0,0], [9E9, 9E9, 9E9, 9E9, 9E9, 9E9]];
	VAR robtarget OpenholeUD_649 := [[395.5, -15.9, 182.88], [-0.175756, 0.684916, 0.689026, 0.158883], [0,0,0,0], [9E9, 9E9, 9E9, 9E9, 9E9, 9E9]];
	VAR robtarget OpenholeUD_650 := [[389.35, -15.9, 183.07], [-0.191139, 0.680783, 0.685185, 0.174703], [0,0,0,0], [9E9, 9E9, 9E9, 9E9, 9E9, 9E9]];
	VAR robtarget OpenholeUD_651 := [[385.35, -15.9, 183.08], [-0.183051, 0.683002, 0.683002, 0.183051], [0,0,0,0], [9E9, 9E9, 9E9, 9E9, 9E9, 9E9]];
	VAR robtarget OpenholeUD_652 := [[381.35, -15.9, 183.09], [-0.183051, 0.683002, 0.683002, 0.183051], [0,0,0,0], [9E9, 9E9, 9E9, 9E9, 9E9, 9E9]];
	VAR robtarget OpenholeUD_653 := [[377.35, -15.9, 183.1], [-0.183051, 0.683002, 0.683002, 0.183051], [0,0,0,0], [9E9, 9E9, 9E9, 9E9, 9E9, 9E9]];
	VAR robtarget OpenholeUD_654 := [[369.35, -15.9, 183.13], [-0.183051, 0.683002, 0.683002, 0.183051], [0,0,0,0], [9E9, 9E9, 9E9, 9E9, 9E9, 9E9]];
	VAR robtarget OpenholeUD_655 := [[369.35, -15.9, 183.13], [-0.183051, 0.683002, 0.683002, 0.183051], [0,0,0,0], [9E9, 9E9, 9E9, 9E9, 9E9, 9E9]];
	VAR robtarget OpenholeUD_656 := [[369.35, -14.7, 183.82], [-0.183051, 0.683002, 0.683002, 0.183051], [0,0,0,0], [9E9, 9E9, 9E9, 9E9, 9E9, 9E9]];
	VAR robtarget OpenholeUD_657 := [[373.35, -14.7, 183.81], [-0.183051, 0.683002, 0.683002, 0.183051], [0,0,0,0], [9E9, 9E9, 9E9, 9E9, 9E9, 9E9]];
	VAR robtarget OpenholeUD_658 := [[377.35, -14.7, 183.8], [-0.183051, 0.683002, 0.683002, 0.183051], [0,0,0,0], [9E9, 9E9, 9E9, 9E9, 9E9, 9E9]];
	VAR robtarget OpenholeUD_659 := [[381.35, -14.7, 183.79], [-0.183051, 0.683002, 0.683002, 0.183051], [0,0,0,0], [9E9, 9E9, 9E9, 9E9, 9E9, 9E9]];
	VAR robtarget OpenholeUD_660 := [[389.35, -14.7, 183.76], [-0.194539, 0.67982, 0.68605, 0.171275], [0,0,0,0], [9E9, 9E9, 9E9, 9E9, 9E9, 9E9]];
	VAR robtarget OpenholeUD_661 := [[393.35, -14.7, 183.59], [-0.184713, 0.682555, 0.688528, 0.161024], [0,0,0,0], [9E9, 9E9, 9E9, 9E9, 9E9, 9E9]];
	VAR robtarget OpenholeUD_662 := [[397.35, -14.7, 183.43], [-0.174516, 0.685233, 0.690924, 0.150411], [0,0,0,0], [9E9, 9E9, 9E9, 9E9, 9E9, 9E9]];
	VAR robtarget OpenholeUD_663 := [[401.34, -14.7, 183.26], [-0.163948, 0.687838, 0.693222, 0.139441], [0,0,0,0], [9E9, 9E9, 9E9, 9E9, 9E9, 9E9]];
	VAR robtarget OpenholeUD_664 := [[405.34, -14.7, 183.09], [-0.153014, 0.690353, 0.695403, 0.128121], [0,0,0,0], [9E9, 9E9, 9E9, 9E9, 9E9, 9E9]];
	VAR robtarget OpenholeUD_665 := [[409.34, -14.7, 182.93], [-0.14172, 0.692759, 0.69745, 0.116461], [0,0,0,0], [9E9, 9E9, 9E9, 9E9, 9E9, 9E9]];
	VAR robtarget OpenholeUD_666 := [[413.33, -14.7, 182.76], [-0.13008, 0.695039, 0.699346, 0.104476], [0,0,0,0], [9E9, 9E9, 9E9, 9E9, 9E9, 9E9]];
	VAR robtarget OpenholeUD_667 := [[417.33, -14.7, 182.59], [-0.118107, 0.697173, 0.701072, 0.092185], [0,0,0,0], [9E9, 9E9, 9E9, 9E9, 9E9, 9E9]];
	VAR robtarget OpenholeUD_668 := [[421.33, -14.7, 182.43], [-0.105823, 0.699143, 0.702611, 0.079611], [0,0,0,0], [9E9, 9E9, 9E9, 9E9, 9E9, 9E9]];
	VAR robtarget OpenholeUD_669 := [[425.32, -14.7, 182.26], [-0.09325, 0.700931, 0.703946, 0.06678], [0,0,0,0], [9E9, 9E9, 9E9, 9E9, 9E9, 9E9]];
	VAR robtarget OpenholeUD_670 := [[429.32, -14.7, 182.1], [-0.080417, 0.702519, 0.705063, 0.053724], [0,0,0,0], [9E9, 9E9, 9E9, 9E9, 9E9, 9E9]];
	VAR robtarget OpenholeUD_671 := [[433.32, -14.7, 181.93], [-0.067356, 0.703891, 0.705947, 0.040478], [0,0,0,0], [9E9, 9E9, 9E9, 9E9, 9E9, 9E9]];
	VAR robtarget OpenholeUD_672 := [[437.31, -14.7, 181.76], [-0.054104, 0.705034, 0.706588, 0.02708], [0,0,0,0], [9E9, 9E9, 9E9, 9E9, 9E9, 9E9]];
	VAR robtarget OpenholeUD_673 := [[444.22, -14.7, 181.47], [-0.03085, 0.706433, 0.707097, 0.003673], [0,0,0,0], [9E9, 9E9, 9E9, 9E9, 9E9, 9E9]];
	VAR robtarget OpenholeUD_674 := [[444.22, -14.7, 181.47], [-0.03085, 0.706433, 0.707097, 0.003673], [0,0,0,0], [9E9, 9E9, 9E9, 9E9, 9E9, 9E9]];
	VAR robtarget OpenholeUD_675 := [[445.45, -13.5, 181.47], [-0.030775, 0.706437, 0.707092, -0.004559], [0,0,0,0], [9E9, 9E9, 9E9, 9E9, 9E9, 9E9]];
	VAR robtarget OpenholeUD_676 := [[441.45, -13.5, 181.68], [-0.044274, 0.705719, 0.707049, 0.009022], [0,0,0,0], [9E9, 9E9, 9E9, 9E9, 9E9, 9E9]];
	VAR robtarget OpenholeUD_677 := [[437.46, -13.5, 181.89], [-0.057657, 0.704752, 0.706747, 0.022545], [0,0,0,0], [9E9, 9E9, 9E9, 9E9, 9E9, 9E9]];
	VAR robtarget OpenholeUD_678 := [[433.46, -13.5, 182.11], [-0.070882, 0.703545, 0.706192, 0.035965], [0,0,0,0], [9E9, 9E9, 9E9, 9E9, 9E9, 9E9]];
	VAR robtarget OpenholeUD_679 := [[429.47, -13.5, 182.32], [-0.083911, 0.70211, 0.70539, 0.049241], [0,0,0,0], [9E9, 9E9, 9E9, 9E9, 9E9, 9E9]];
	VAR robtarget OpenholeUD_680 := [[425.47, -13.5, 182.53], [-0.096707, 0.700463, 0.704354, 0.062334], [0,0,0,0], [9E9, 9E9, 9E9, 9E9, 9E9, 9E9]];
	VAR robtarget OpenholeUD_681 := [[421.48, -13.5, 182.74], [-0.109238, 0.698618, 0.703096, 0.07521], [0,0,0,0], [9E9, 9E9, 9E9, 9E9, 9E9, 9E9]];
	VAR robtarget OpenholeUD_682 := [[417.49, -13.5, 182.96], [-0.121478, 0.696594, 0.70163, 0.087836], [0,0,0,0], [9E9, 9E9, 9E9, 9E9, 9E9, 9E9]];
	VAR robtarget OpenholeUD_683 := [[413.49, -13.5, 183.17], [-0.133402, 0.694409, 0.699974, 0.100185], [0,0,0,0], [9E9, 9E9, 9E9, 9E9, 9E9, 9E9]];
	VAR robtarget OpenholeUD_684 := [[409.5, -13.5, 183.38], [-0.144991, 0.692082, 0.698143, 0.112232], [0,0,0,0], [9E9, 9E9, 9E9, 9E9, 9E9, 9E9]];
	VAR robtarget OpenholeUD_685 := [[405.5, -13.5, 183.59], [-0.156231, 0.689632, 0.696157, 0.12396], [0,0,0,0], [9E9, 9E9, 9E9, 9E9, 9E9, 9E9]];
